LIN {X 0,Y 312.008,Z 393.675,A -85,B 0,C 180,E1 -15970.642,E2 -15970.642} C_VEL
LIN {X 0,Y 309.951,Z 389.912,A -85,B 0,C 180,E1 -15971.165,E2 -15971.165} C_VEL
LIN {X 0,Y 307.208,Z 381.469,A -85,B 0,C 180,E1 -15974.218,E2 -15974.218} C_VEL
LIN {X 0,Y 305.411,Z 376.065,A -85,B 0,C 180,E1 -15976.343,E2 -15976.343} C_VEL
LIN {X 0,Y 305.408,Z 376.064,A -85,B 0,C 180,E1 -15979.885,E2 -15979.885} C_VEL
LIN {X 0,Y 305.462,Z 376.035,A -85,B 0,C 180,E1 -15983.637,E2 -15983.637} C_VEL
LIN {X 0,Y 305.464,Z 376.059,A -85,B 0,C 180,E1 -15986.484,E2 -15986.484} C_VEL
LIN {X 0,Y 305.432,Z 376.032,A -85,B 0,C 180,E1 -15989.588,E2 -15989.588} C_VEL
LIN {X 0,Y 305.466,Z 376.057,A -85,B 0,C 180,E1 -15992.604,E2 -15992.604} C_VEL
LIN {X 0,Y 305.486,Z 376.057,A -85,B 0,C 180,E1 -15995.537,E2 -15995.537} C_VEL
LIN {X 0,Y 305.511,Z 376.05,A -85,B 0,C 180,E1 -15999.815,E2 -15999.815} C_VEL
LIN {X 0,Y 305.575,Z 376.046,A -85,B 0,C 180,E1 -16002.604,E2 -16002.604} C_VEL
LIN {X 0,Y 305.65,Z 376.036,A -85,B 0,C 180,E1 -16005.35,E2 -16005.35} C_VEL
LIN {X 0,Y 305.625,Z 376.039,A -85,B 0,C 180,E1 -16009.4,E2 -16009.4} C_VEL
LIN {X 0,Y 305.747,Z 376.015,A -85,B 0,C 180,E1 -16012.073,E2 -16012.073} C_VEL
LIN {X 0,Y 305.667,Z 376.028,A -85,B 0,C 180,E1 -16014.724,E2 -16014.724} C_VEL
LIN {X 0,Y 305.941,Z 375.994,A -85,B 0,C 180,E1 -16018.684,E2 -16018.684} C_VEL
LIN {X 0,Y 305.949,Z 376,A -85,B 0,C 180,E1 -16021.317,E2 -16021.317} C_VEL
LIN {X 0,Y 305.789,Z 376.012,A -85,B 0,C 180,E1 -16026.599,E2 -16026.599} C_VEL
LIN {X 0,Y 305.7,Z 376.031,A -85,B 0,C 180,E1 -16029.261,E2 -16029.261} C_VEL
LIN {X 0,Y 305.592,Z 376.043,A -85,B 0,C 180,E1 -16033.297,E2 -16033.297} C_VEL
LIN {X 0,Y 305.596,Z 376.042,A -85,B 0,C 180,E1 -16036.021,E2 -16036.021} C_VEL
LIN {X 0,Y 305.563,Z 376.014,A -85,B 0,C 180,E1 -16039.437,E2 -16039.437} C_VEL
LIN {X 0,Y 305.457,Z 376.061,A -85,B 0,C 180,E1 -16043.026,E2 -16043.026} C_VEL
LIN {X 0,Y 305.459,Z 376.033,A -85,B 0,C 180,E1 -16046.193,E2 -16046.193} C_VEL
LIN {X 0,Y 305.465,Z 376.058,A -85,B 0,C 180,E1 -16049.039,E2 -16049.039} C_VEL
LIN {X 0,Y 305.439,Z 376.045,A -85,B 0,C 180,E1 -16051.953,E2 -16051.953} C_VEL
LIN {X 0,Y 305.463,Z 376.042,A -85,B 0,C 180,E1 -16055.114,E2 -16055.114} C_VEL
LIN {X 0,Y 305.458,Z 376.146,A -85,B 0,C 180,E1 -16057.778,E2 -16057.778} C_VEL
LIN {X 0,Y 305.692,Z 377.224,A -85,B 0,C 180,E1 -16058.109,E2 -16058.109} C_VEL
LIN {X 0,Y 307.128,Z 379.845,A -85,B 0,C 180,E1 -16058.474,E2 -16058.474} C_VEL
LIN {X 0,Y 309.196,Z 382.473,A -85,B 0,C 180,E1 -16058.952,E2 -16058.952} C_VEL
LIN {X 0,Y 315.262,Z 391.574,A -85,B 0,C 180,E1 -16060.337,E2 -16060.337} C_VEL
LIN {X 0,Y 323.299,Z 404.841,A -85,B 0,C 180,E1 -16062.079,E2 -16062.079} C_VEL
LIN {X 0,Y 331.219,Z 419.433,A -85,B 0,C 180,E1 -16063.71,E2 -16063.71} C_VEL
LIN {X 0,Y 336.796,Z 430.906,A -85,B 0,C 180,E1 -16064.82,E2 -16064.82} C_VEL
LIN {X 0,Y 332.896,Z 525.367,A -85,B 0,C 180,E1 -16066.831,E2 -16066.831} C_VEL
LIN {X 0,Y 332.024,Z 544.302,A -85,B 0,C 180,E1 -16067.312,E2 -16067.312} C_VEL
LIN {X 0,Y 330.677,Z 559.768,A -85,B 0,C 180,E1 -16067.932,E2 -16067.932} C_VEL
LIN {X 0,Y 329.028,Z 573.938,A -85,B 0,C 180,E1 -16068.739,E2 -16068.739} C_VEL
LIN {X 0,Y 326.677,Z 588.476,A -85,B 0,C 180,E1 -16069.804,E2 -16069.804} C_VEL
LIN {X 0,Y 324.399,Z 601.799,A -85,B 0,C 180,E1 -16071.077,E2 -16071.077} C_VEL
LIN {X 0,Y 321.786,Z 614.094,A -85,B 0,C 180,E1 -16072.497,E2 -16072.497} C_VEL
LIN {X 0,Y 319.107,Z 625.525,A -85,B 0,C 180,E1 -16074.099,E2 -16074.099} C_VEL
LIN {X 0,Y 316.387,Z 636.114,A -85,B 0,C 180,E1 -16075.889,E2 -16075.889} C_VEL
LIN {X 0,Y 313.466,Z 647.104,A -85,B 0,C 180,E1 -16078.154,E2 -16078.154} C_VEL
LIN {X 0,Y 310.816,Z 656.515,A -85,B 0,C 180,E1 -16080.541,E2 -16080.541} C_VEL
LIN {X 0,Y 308.727,Z 664.118,A -85,B 0,C 180,E1 -16082.916,E2 -16082.916} C_VEL
LIN {X 0,Y 306.792,Z 671.137,A -85,B 0,C 180,E1 -16085.648,E2 -16085.648} C_VEL
LIN {X 0,Y 305.382,Z 676.578,A -85,B 0,C 180,E1 -16088.394,E2 -16088.394} C_VEL
LIN {X 0,Y 304.506,Z 680.595,A -85,B 0,C 180,E1 -16091.148,E2 -16091.148} C_VEL
LIN {X 0,Y 303.877,Z 683.314,A -85,B 0,C 180,E1 -16093.887,E2 -16093.887} C_VEL
LIN {X 0,Y 303.662,Z 684.816,A -85,B 0,C 180,E1 -16096.618,E2 -16096.618} C_VEL
LIN {X 0,Y 303.427,Z 685.154,A -85,B 0,C 180,E1 -16099.322,E2 -16099.322} C_VEL
LIN {X 0,Y 303.481,Z 684.345,A -85,B 0,C 180,E1 -16102.013,E2 -16102.013} C_VEL
LIN {X 0,Y 303.749,Z 682.375,A -85,B 0,C 180,E1 -16104.69,E2 -16104.69} C_VEL
LIN {X 0,Y 303.979,Z 679.192,A -85,B 0,C 180,E1 -16107.35,E2 -16107.35} C_VEL
LIN {X 0,Y 304.483,Z 674.772,A -85,B 0,C 180,E1 -16110,E2 -16110} C_VEL
LIN {X 0,Y 305.284,Z 669.021,A -85,B 0,C 180,E1 -16112.639,E2 -16112.639} C_VEL
LIN {X 0,Y 306.568,Z 661.77,A -85,B 0,C 180,E1 -16115.261,E2 -16115.261} C_VEL
LIN {X 0,Y 308.121,Z 654.006,A -85,B 0,C 180,E1 -16117.536,E2 -16117.536} C_VEL
LIN {X 0,Y 309.891,Z 644.712,A -85,B 0,C 180,E1 -16119.793,E2 -16119.793} C_VEL
LIN {X 0,Y 311.707,Z 635.269,A -85,B 0,C 180,E1 -16121.708,E2 -16121.708} C_VEL
LIN {X 0,Y 313.915,Z 624.043,A -85,B 0,C 180,E1 -16123.596,E2 -16123.596} C_VEL
LIN {X 0,Y 315.97,Z 611.759,A -85,B 0,C 180,E1 -16125.315,E2 -16125.315} C_VEL
LIN {X 0,Y 318.171,Z 598.17,A -85,B 0,C 180,E1 -16126.853,E2 -16126.853} C_VEL
LIN {X 0,Y 319.993,Z 584.854,A -85,B 0,C 180,E1 -16128.073,E2 -16128.073} C_VEL
LIN {X 0,Y 321.678,Z 570.085,A -85,B 0,C 180,E1 -16129.131,E2 -16129.131} C_VEL
LIN {X 0,Y 323.055,Z 555.393,A -85,B 0,C 180,E1 -16129.914,E2 -16129.914} C_VEL
LIN {X 0,Y 323.925,Z 540.407,A -85,B 0,C 180,E1 -16130.479,E2 -16130.479} C_VEL
LIN {X 0,Y 327.674,Z 425.087,A -85,B 0,C 180,E1 -16133.005,E2 -16133.005} C_VEL
LIN {X 0,Y 327.355,Z 423.116,A -85,B 0,C 180,E1 -16133.086,E2 -16133.086} C_VEL
LIN {X 0,Y 319.54,Z 404.611,A -85,B 0,C 180,E1 -16134.363,E2 -16134.363} C_VEL
LIN {X 0,Y 311.06,Z 386.835,A -85,B 0,C 180,E1 -16135.777,E2 -16135.777} C_VEL
LIN {X 0,Y 306.672,Z 379.243,A -85,B 0,C 180,E1 -16136.503,E2 -16136.503} C_VEL
LIN {X 0,Y 305.851,Z 377.64,A -85,B 0,C 180,E1 -16136.647,E2 -16136.647} C_VEL
LIN {X 0,Y 305.049,Z 376.531,A -85,B 0,C 180,E1 -16136.872,E2 -16136.872} C_VEL
LIN {X 0,Y 303.78,Z 376.27,A -85,B 0,C 180,E1 -16137.343,E2 -16137.343} C_VEL
LIN {X 0,Y 300.721,Z 376.645,A -85,B 0,C 180,E1 -16139.038,E2 -16139.038} C_VEL
LIN {X 0,Y 299.352,Z 377.162,A -85,B 0,C 180,E1 -16140.301,E2 -16140.301} C_VEL
LIN {X 0,Y 298.388,Z 376.931,A -85,B 0,C 180,E1 -16142.464,E2 -16142.464} C_VEL
LIN {X 0,Y 298.409,Z 376.927,A -85,B 0,C 180,E1 -16146.071,E2 -16146.071} C_VEL
LIN {X 0,Y 298.377,Z 376.934,A -85,B 0,C 180,E1 -16149.491,E2 -16149.491} C_VEL
LIN {X 0,Y 298.403,Z 376.94,A -85,B 0,C 180,E1 -16153.103,E2 -16153.103} C_VEL
LIN {X 0,Y 298.374,Z 376.928,A -85,B 0,C 180,E1 -16156.915,E2 -16156.915} C_VEL
LIN {X 0,Y 298.354,Z 376.938,A -85,B 0,C 180,E1 -16161.019,E2 -16161.019} C_VEL
LIN {X 0,Y 298.407,Z 376.939,A -85,B 0,C 180,E1 -16163.928,E2 -16163.928} C_VEL
LIN {X 0,Y 298.396,Z 376.937,A -85,B 0,C 180,E1 -16167.199,E2 -16167.199} C_VEL
LIN {X 0,Y 298.404,Z 376.927,A -85,B 0,C 180,E1 -16170.625,E2 -16170.625} C_VEL
LIN {X 0,Y 298.416,Z 376.89,A -85,B 0,C 180,E1 -16174.917,E2 -16174.917} C_VEL
LIN {X 0,Y 298.429,Z 376.937,A -85,B 0,C 180,E1 -16179.313,E2 -16179.313} C_VEL
LIN {X 0,Y 298.508,Z 376.909,A -85,B 0,C 180,E1 -16182.177,E2 -16182.177} C_VEL
LIN {X 0,Y 298.588,Z 376.913,A -85,B 0,C 180,E1 -16184.994,E2 -16184.994} C_VEL
LIN {X 0,Y 298.586,Z 376.897,A -85,B 0,C 180,E1 -16189.146,E2 -16189.146} C_VEL
LIN {X 0,Y 298.7,Z 376.901,A -85,B 0,C 180,E1 -16191.884,E2 -16191.884} C_VEL
LIN {X 0,Y 298.63,Z 376.893,A -85,B 0,C 180,E1 -16194.598,E2 -16194.598} C_VEL
LIN {X 0,Y 298.915,Z 376.873,A -85,B 0,C 180,E1 -16198.652,E2 -16198.652} C_VEL
LIN {X 0,Y 298.909,Z 376.859,A -85,B 0,C 180,E1 -16201.347,E2 -16201.347} C_VEL
LIN {X 0,Y 298.635,Z 376.912,A -85,B 0,C 180,E1 -16205.401,E2 -16205.401} C_VEL
LIN {X 0,Y 298.709,Z 376.893,A -85,B 0,C 180,E1 -16208.819,E2 -16208.819} C_VEL
LIN {X 0,Y 298.545,Z 376.911,A -85,B 0,C 180,E1 -16212.231,E2 -16212.231} C_VEL
LIN {X 0,Y 298.524,Z 376.92,A -85,B 0,C 180,E1 -16215.15,E2 -16215.15} C_VEL
LIN {X 0,Y 298.499,Z 376.923,A -85,B 0,C 180,E1 -16219.647,E2 -16219.647} C_VEL
LIN {X 0,Y 298.424,Z 376.932,A -85,B 0,C 180,E1 -16223.6,E2 -16223.6} C_VEL
LIN {X 0,Y 298.408,Z 376.931,A -85,B 0,C 180,E1 -16226.582,E2 -16226.582} C_VEL
LIN {X 0,Y 298.394,Z 376.936,A -85,B 0,C 180,E1 -16229.643,E2 -16229.643} C_VEL
LIN {X 0,Y 298.392,Z 376.937,A -85,B 0,C 180,E1 -16232.8,E2 -16232.8} C_VEL
LIN {X 0,Y 298.426,Z 376.935,A -85,B 0,C 180,E1 -16236.802,E2 -16236.802} C_VEL
LIN {X 0,Y 298.347,Z 376.945,A -85,B 0,C 180,E1 -16241.267,E2 -16241.267} C_VEL
LIN {X 0,Y 298.353,Z 376.946,A -85,B 0,C 180,E1 -16245.034,E2 -16245.034} C_VEL
LIN {X 0,Y 298.378,Z 377.05,A -85,B 0,C 180,E1 -16248.765,E2 -16248.765} C_VEL
LIN {X 0,Y 301.352,Z 387.503,A -85,B 0,C 180,E1 -16251.914,E2 -16251.914} C_VEL
LIN {X 0,Y 302.25,Z 391.009,A -85,B 0,C 180,E1 -16252.878,E2 -16252.878} C_VEL
LIN {X 0,Y 310.107,Z 407.933,A -85,B 0,C 180,E1 -16254.276,E2 -16254.276} C_VEL
LIN {X 0,Y 317.769,Z 426.003,A -85,B 0,C 180,E1 -16255.596,E2 -16255.596} C_VEL
LIN {X 0,Y 318.599,Z 429.317,A -85,B 0,C 180,E1 -16255.77,E2 -16255.77} C_VEL
LIN {X 0,Y 321.034,Z 444.923,A -85,B 0,C 180,E1 -16256.421,E2 -16256.421} C_VEL
LIN {X 0,Y 317.296,Z 558.27,A -85,B 0,C 180,E1 -16258.957,E2 -16258.957} C_VEL
LIN {X 0,Y 316.142,Z 573.476,A -85,B 0,C 180,E1 -16259.527,E2 -16259.527} C_VEL
LIN {X 0,Y 314.609,Z 587.681,A -85,B 0,C 180,E1 -16260.288,E2 -16260.288} C_VEL
LIN {X 0,Y 312.776,Z 601.94,A -85,B 0,C 180,E1 -16261.309,E2 -16261.309} C_VEL
LIN {X 0,Y 310.741,Z 615.574,A -85,B 0,C 180,E1 -16262.56,E2 -16262.56} C_VEL
LIN {X 0,Y 308.581,Z 628.233,A -85,B 0,C 180,E1 -16263.997,E2 -16263.997} C_VEL
LIN {X 0,Y 306.139,Z 641.062,A -85,B 0,C 180,E1 -16265.773,E2 -16265.773} C_VEL
LIN {X 0,Y 304.1,Z 651.792,A -85,B 0,C 180,E1 -16267.582,E2 -16267.582} C_VEL
LIN {X 0,Y 302.25,Z 661.737,A -85,B 0,C 180,E1 -16269.587,E2 -16269.587} C_VEL
LIN {X 0,Y 300.332,Z 671.446,A -85,B 0,C 180,E1 -16271.937,E2 -16271.937} C_VEL
LIN {X 0,Y 298.89,Z 679.527,A -85,B 0,C 180,E1 -16274.312,E2 -16274.312} C_VEL
LIN {X 0,Y 297.746,Z 687.046,A -85,B 0,C 180,E1 -16277.042,E2 -16277.042} C_VEL
LIN {X 0,Y 296.974,Z 692.994,A -85,B 0,C 180,E1 -16279.776,E2 -16279.776} C_VEL
LIN {X 0,Y 296.719,Z 696.522,A -85,B 0,C 180,E1 -16281.83,E2 -16281.83} C_VEL
LIN {X 0,Y 296.549,Z 700.073,A -85,B 0,C 180,E1 -16284.56,E2 -16284.56} C_VEL
LIN {X 0,Y 296.54,Z 702.389,A -85,B 0,C 180,E1 -16287.283,E2 -16287.283} C_VEL
LIN {X 0,Y 296.533,Z 703.529,A -85,B 0,C 180,E1 -16290,E2 -16290} C_VEL
LIN {X 0,Y 296.525,Z 703.493,A -85,B 0,C 180,E1 -16292.717,E2 -16292.717} C_VEL
LIN {X 0,Y 296.51,Z 702.276,A -85,B 0,C 180,E1 -16295.44,E2 -16295.44} C_VEL
LIN {X 0,Y 296.704,Z 699.922,A -85,B 0,C 180,E1 -16298.171,E2 -16298.171} C_VEL
LIN {X 0,Y 297.218,Z 696.389,A -85,B 0,C 180,E1 -16300.904,E2 -16300.904} C_VEL
LIN {X 0,Y 298.236,Z 691.598,A -85,B 0,C 180,E1 -16303.63,E2 -16303.63} C_VEL
LIN {X 0,Y 299.688,Z 685.423,A -85,B 0,C 180,E1 -16306.345,E2 -16306.345} C_VEL
LIN {X 0,Y 301.786,Z 677.699,A -85,B 0,C 180,E1 -16309.028,E2 -16309.028} C_VEL
LIN {X 0,Y 304.1,Z 669.495,A -85,B 0,C 180,E1 -16311.346,E2 -16311.346} C_VEL
LIN {X 0,Y 306.627,Z 660.122,A -85,B 0,C 180,E1 -16313.536,E2 -16313.536} C_VEL
LIN {X 0,Y 309.527,Z 649.618,A -85,B 0,C 180,E1 -16315.557,E2 -16315.557} C_VEL
LIN {X 0,Y 312.649,Z 637.725,A -85,B 0,C 180,E1 -16317.44,E2 -16317.44} C_VEL
LIN {X 0,Y 315.537,Z 625.876,A -85,B 0,C 180,E1 -16318.976,E2 -16318.976} C_VEL
LIN {X 0,Y 318.347,Z 613.086,A -85,B 0,C 180,E1 -16320.331,E2 -16320.331} C_VEL
LIN {X 0,Y 320.902,Z 599.132,A -85,B 0,C 180,E1 -16321.527,E2 -16321.527} C_VEL
LIN {X 0,Y 323.175,Z 584.768,A -85,B 0,C 180,E1 -16322.471,E2 -16322.471} C_VEL
LIN {X 0,Y 325.045,Z 570.002,A -85,B 0,C 180,E1 -16323.182,E2 -16323.182} C_VEL
LIN {X 0,Y 326.354,Z 554.891,A -85,B 0,C 180,E1 -16323.678,E2 -16323.678} C_VEL
LIN {X 0,Y 330.69,Z 446.764,A -85,B 0,C 180,E1 -16326.074,E2 -16326.074} C_VEL
LIN {X 0,Y 329.355,Z 439.216,A -85,B 0,C 180,E1 -16326.478,E2 -16326.478} C_VEL
LIN {X 0,Y 321.063,Z 421.84,A -85,B 0,C 180,E1 -16328.245,E2 -16328.245} C_VEL
LIN {X 0,Y 312.778,Z 406.54,A -85,B 0,C 180,E1 -16330.1,E2 -16330.1} C_VEL
LIN {X 0,Y 307.454,Z 397.794,A -85,B 0,C 180,E1 -16331.344,E2 -16331.344} C_VEL
LIN {X 0,Y 305.141,Z 394.014,A -85,B 0,C 180,E1 -16331.907,E2 -16331.907} C_VEL
LIN {X 0,Y 302.575,Z 389.595,A -85,B 0,C 180,E1 -16332.584,E2 -16332.584} C_VEL
LIN {X 0,Y 299.446,Z 380.298,A -85,B 0,C 180,E1 -16336.184,E2 -16336.184} C_VEL
LIN {X 0,Y 298.4,Z 376.939,A -85,B 0,C 180,E1 -16337.61,E2 -16337.61} C_VEL
LIN {X 0,Y 298.384,Z 376.941,A -85,B 0,C 180,E1 -16341.011,E2 -16341.011} C_VEL
LIN {X 0,Y 298.404,Z 376.913,A -85,B 0,C 180,E1 -16343.929,E2 -16343.929} C_VEL
LIN {X 0,Y 298.392,Z 376.931,A -85,B 0,C 180,E1 -16347.2,E2 -16347.2} C_VEL
LIN {X 0,Y 298.407,Z 376.917,A -85,B 0,C 180,E1 -16350.624,E2 -16350.624} C_VEL
LIN {X 0,Y 298.446,Z 376.934,A -85,B 0,C 180,E1 -16354.921,E2 -16354.921} C_VEL
LIN {X 0,Y 298.444,Z 376.933,A -85,B 0,C 180,E1 -16359.315,E2 -16359.315} C_VEL
LIN {X 0,Y 298.535,Z 376.924,A -85,B 0,C 180,E1 -16362.18,E2 -16362.18} C_VEL
LIN {X 0,Y 298.594,Z 376.911,A -85,B 0,C 180,E1 -16364.995,E2 -16364.995} C_VEL
LIN {X 0,Y 298.584,Z 376.917,A -85,B 0,C 180,E1 -16369.147,E2 -16369.147} C_VEL
LIN {X 0,Y 298.699,Z 376.892,A -85,B 0,C 180,E1 -16371.885,E2 -16371.885} C_VEL
LIN {X 0,Y 298.636,Z 376.905,A -85,B 0,C 180,E1 -16374.599,E2 -16374.599} C_VEL
LIN {X 0,Y 298.91,Z 376.87,A -85,B 0,C 180,E1 -16378.653,E2 -16378.653} C_VEL
LIN {X 0,Y 298.916,Z 376.876,A -85,B 0,C 180,E1 -16381.348,E2 -16381.348} C_VEL
LIN {X 0,Y 298.737,Z 376.889,A -85,B 0,C 180,E1 -16386.756,E2 -16386.756} C_VEL
LIN {X 0,Y 298.632,Z 376.911,A -85,B 0,C 180,E1 -16389.483,E2 -16389.483} C_VEL
LIN {X 0,Y 298.555,Z 376.92,A -85,B 0,C 180,E1 -16393.616,E2 -16393.616} C_VEL
LIN {X 0,Y 298.551,Z 376.923,A -85,B 0,C 180,E1 -16396.409,E2 -16396.409} C_VEL
LIN {X 0,Y 298.496,Z 376.893,A -85,B 0,C 180,E1 -16399.646,E2 -16399.646} C_VEL
LIN {X 0,Y 298.386,Z 376.936,A -85,B 0,C 180,E1 -16403.604,E2 -16403.604} C_VEL
LIN {X 0,Y 298.407,Z 376.913,A -85,B 0,C 180,E1 -16406.583,E2 -16406.583} C_VEL
LIN {X 0,Y 298.402,Z 376.926,A -85,B 0,C 180,E1 -16409.644,E2 -16409.644} C_VEL
LIN {X 0,Y 298.395,Z 376.935,A -85,B 0,C 180,E1 -16412.801,E2 -16412.801} C_VEL
LIN {X 0,Y 298.418,Z 376.96,A -85,B 0,C 180,E1 -16416.53,E2 -16416.53} C_VEL
LIN {X 0,Y 298.525,Z 377.581,A -85,B 0,C 180,E1 -16416.669,E2 -16416.669} C_VEL
LIN {X 0,Y 299.706,Z 380.222,A -85,B 0,C 180,E1 -16417.009,E2 -16417.009} C_VEL
LIN {X 0,Y 301.827,Z 382.507,A -85,B 0,C 180,E1 -16417.521,E2 -16417.521} C_VEL
LIN {X 0,Y 303.801,Z 385.631,A -85,B 0,C 180,E1 -16418.021,E2 -16418.021} C_VEL
LIN {X 0,Y 305.3,Z 387.534,A -85,B 0,C 180,E1 -16418.377,E2 -16418.377} C_VEL
LIN {X 0,Y 311.863,Z 397.674,A -85,B 0,C 180,E1 -16419.928,E2 -16419.928} C_VEL
LIN {X 0,Y 319.09,Z 409.756,A -85,B 0,C 180,E1 -16421.543,E2 -16421.543} C_VEL
LIN {X 0,Y 326.096,Z 422.733,A -85,B 0,C 180,E1 -16423.036,E2 -16423.036} C_VEL
LIN {X 0,Y 331.26,Z 433.44,A -85,B 0,C 180,E1 -16424.107,E2 -16424.107} C_VEL
LIN {X 0,Y 327.037,Z 530.162,A -85,B 0,C 180,E1 -16426.181,E2 -16426.181} C_VEL
LIN {X 0,Y 326.245,Z 546.715,A -85,B 0,C 180,E1 -16426.652,E2 -16426.652} C_VEL
LIN {X 0,Y 324.83,Z 561.215,A -85,B 0,C 180,E1 -16427.262,E2 -16427.262} C_VEL
LIN {X 0,Y 323.026,Z 575.6,A -85,B 0,C 180,E1 -16428.113,E2 -16428.113} C_VEL
LIN {X 0,Y 320.758,Z 588.911,A -85,B 0,C 180,E1 -16429.112,E2 -16429.112} C_VEL
LIN {X 0,Y 318.366,Z 602.299,A -85,B 0,C 180,E1 -16430.416,E2 -16430.416} C_VEL
LIN {X 0,Y 315.67,Z 614.443,A -85,B 0,C 180,E1 -16431.843,E2 -16431.843} C_VEL
LIN {X 0,Y 312.879,Z 625.846,A -85,B 0,C 180,E1 -16433.469,E2 -16433.469} C_VEL
LIN {X 0,Y 309.822,Z 637.27,A -85,B 0,C 180,E1 -16435.452,E2 -16435.452} C_VEL
LIN {X 0,Y 307.14,Z 646.858,A -85,B 0,C 180,E1 -16437.472,E2 -16437.472} C_VEL
LIN {X 0,Y 304.374,Z 656.187,A -85,B 0,C 180,E1 -16439.854,E2 -16439.854} C_VEL
LIN {X 0,Y 302.142,Z 663.872,A -85,B 0,C 180,E1 -16442.276,E2 -16442.276} C_VEL
LIN {X 0,Y 300.05,Z 670.989,A -85,B 0,C 180,E1 -16445.064,E2 -16445.064} C_VEL
LIN {X 0,Y 298.521,Z 676.514,A -85,B 0,C 180,E1 -16447.872,E2 -16447.872} C_VEL
LIN {X 0,Y 297.484,Z 680.892,A -85,B 0,C 180,E1 -16450.91,E2 -16450.91} C_VEL
LIN {X 0,Y 296.846,Z 683.406,A -85,B 0,C 180,E1 -16453.495,E2 -16453.495} C_VEL
LIN {X 0,Y 296.569,Z 684.991,A -85,B 0,C 180,E1 -16456.317,E2 -16456.317} C_VEL
LIN {X 0,Y 296.356,Z 685.393,A -85,B 0,C 180,E1 -16459.064,E2 -16459.064} C_VEL
LIN {X 0,Y 296.39,Z 684.656,A -85,B 0,C 180,E1 -16461.821,E2 -16461.821} C_VEL
LIN {X 0,Y 296.648,Z 682.726,A -85,B 0,C 180,E1 -16464.562,E2 -16464.562} C_VEL
LIN {X 0,Y 296.882,Z 679.615,A -85,B 0,C 180,E1 -16467.286,E2 -16467.286} C_VEL
LIN {X 0,Y 297.402,Z 675.273,A -85,B 0,C 180,E1 -16470,E2 -16470} C_VEL
LIN {X 0,Y 298.221,Z 669.604,A -85,B 0,C 180,E1 -16472.702,E2 -16472.702} C_VEL
LIN {X 0,Y 299.523,Z 662.443,A -85,B 0,C 180,E1 -16475.386,E2 -16475.386} C_VEL
LIN {X 0,Y 301.111,Z 654.778,A -85,B 0,C 180,E1 -16477.713,E2 -16477.713} C_VEL
LIN {X 0,Y 302.956,Z 645.59,A -85,B 0,C 180,E1 -16480.02,E2 -16480.02} C_VEL
LIN {X 0,Y 304.813,Z 636.277,A -85,B 0,C 180,E1 -16481.977,E2 -16481.977} C_VEL
LIN {X 0,Y 307.091,Z 625.19,A -85,B 0,C 180,E1 -16483.904,E2 -16483.904} C_VEL
LIN {X 0,Y 309.222,Z 613.076,A -85,B 0,C 180,E1 -16485.658,E2 -16485.658} C_VEL
LIN {X 0,Y 311.462,Z 599.754,A -85,B 0,C 180,E1 -16487.227,E2 -16487.227} C_VEL
LIN {X 0,Y 313.592,Z 584.865,A -85,B 0,C 180,E1 -16488.624,E2 -16488.624} C_VEL
LIN {X 0,Y 315.309,Z 570.043,A -85,B 0,C 180,E1 -16489.702,E2 -16489.702} C_VEL
LIN {X 0,Y 316.741,Z 555.244,A -85,B 0,C 180,E1 -16490.497,E2 -16490.497} C_VEL
LIN {X 0,Y 317.652,Z 540.071,A -85,B 0,C 180,E1 -16491.071,E2 -16491.071} C_VEL
LIN {X 0,Y 321.482,Z 426.854,A -85,B 0,C 180,E1 -16493.589,E2 -16493.589} C_VEL
LIN {X 0,Y 321.068,Z 424.843,A -85,B 0,C 180,E1 -16493.683,E2 -16493.683} C_VEL
LIN {X 0,Y 313.395,Z 406.641,A -85,B 0,C 180,E1 -16494.983,E2 -16494.983} C_VEL
LIN {X 0,Y 305.579,Z 390.346,A -85,B 0,C 180,E1 -16496.33,E2 -16496.33} C_VEL
LIN {X 0,Y 299.769,Z 380.27,A -85,B 0,C 180,E1 -16497.331,E2 -16497.331} C_VEL
LIN {X 0,Y 298.5,Z 377.502,A -85,B 0,C 180,E1 -16497.573,E2 -16497.573} C_VEL
LIN {X 0,Y 298.421,Z 376.937,A -85,B 0,C 180,E1 -16497.619,E2 -16497.619} C_VEL
LIN {X 0,Y 298.382,Z 376.943,A -85,B 0,C 180,E1 -16501.211,E2 -16501.211} C_VEL
LIN {X 0,Y 298.388,Z 376.931,A -85,B 0,C 180,E1 -16502.464,E2 -16502.464} C_VEL
LIN {X 0,Y 297.729,Z 377.021,A -85,B 0,C 180,E1 -16503.59,E2 -16503.59} C_VEL
LIN {X 0,Y 294.858,Z 377.374,A -85,B 0,C 180,E1 -16505.422,E2 -16505.422} C_VEL
LIN {X 0,Y 292.426,Z 377.674,A -85,B 0,C 180,E1 -16506.909,E2 -16506.909} C_VEL
LIN {X 0,Y 291.398,Z 377.813,A -85,B 0,C 180,E1 -16508.062,E2 -16508.062} C_VEL
LIN {X 0,Y 291.323,Z 377.817,A -85,B 0,C 180,E1 -16508.452,E2 -16508.452} C_VEL
LIN {X 0,Y 291.291,Z 377.824,A -85,B 0,C 180,E1 -16512.498,E2 -16512.498} C_VEL
LIN {X 0,Y 291.292,Z 377.805,A -85,B 0,C 180,E1 -16516.37,E2 -16516.37} C_VEL
LIN {X 0,Y 291.313,Z 377.817,A -85,B 0,C 180,E1 -16520.535,E2 -16520.535} C_VEL
LIN {X 0,Y 291.388,Z 377.812,A -85,B 0,C 180,E1 -16522.916,E2 -16522.916} C_VEL
LIN {X 0,Y 291.346,Z 377.811,A -85,B 0,C 180,E1 -16526.301,E2 -16526.301} C_VEL
LIN {X 0,Y 291.367,Z 377.808,A -85,B 0,C 180,E1 -16530.268,E2 -16530.268} C_VEL
LIN {X 0,Y 291.344,Z 377.764,A -85,B 0,C 180,E1 -16534.264,E2 -16534.264} C_VEL
LIN {X 0,Y 291.354,Z 377.805,A -85,B 0,C 180,E1 -16537.297,E2 -16537.297} C_VEL
LIN {X 0,Y 291.442,Z 377.804,A -85,B 0,C 180,E1 -16540.268,E2 -16540.268} C_VEL
LIN {X 0,Y 291.517,Z 377.793,A -85,B 0,C 180,E1 -16544.652,E2 -16544.652} C_VEL
LIN {X 0,Y 291.532,Z 377.775,A -85,B 0,C 180,E1 -16548.88,E2 -16548.88} C_VEL
LIN {X 0,Y 291.654,Z 377.78,A -85,B 0,C 180,E1 -16551.686,E2 -16551.686} C_VEL
LIN {X 0,Y 291.6,Z 377.769,A -85,B 0,C 180,E1 -16554.467,E2 -16554.467} C_VEL
LIN {X 0,Y 291.881,Z 377.749,A -85,B 0,C 180,E1 -16558.62,E2 -16558.62} C_VEL
LIN {X 0,Y 291.877,Z 377.735,A -85,B 0,C 180,E1 -16561.379,E2 -16561.379} C_VEL
LIN {X 0,Y 291.605,Z 377.786,A -85,B 0,C 180,E1 -16565.532,E2 -16565.532} C_VEL
LIN {X 0,Y 291.668,Z 377.77,A -85,B 0,C 180,E1 -16568.909,E2 -16568.909} C_VEL
LIN {X 0,Y 291.509,Z 377.786,A -85,B 0,C 180,E1 -16572.531,E2 -16572.531} C_VEL
LIN {X 0,Y 291.461,Z 377.801,A -85,B 0,C 180,E1 -16575.381,E2 -16575.381} C_VEL
LIN {X 0,Y 291.452,Z 377.804,A -85,B 0,C 180,E1 -16579.874,E2 -16579.874} C_VEL
LIN {X 0,Y 291.364,Z 377.814,A -85,B 0,C 180,E1 -16584.208,E2 -16584.208} C_VEL
LIN {X 0,Y 291.354,Z 377.813,A -85,B 0,C 180,E1 -16587.278,E2 -16587.278} C_VEL
LIN {X 0,Y 291.319,Z 377.819,A -85,B 0,C 180,E1 -16590.438,E2 -16590.438} C_VEL
LIN {X 0,Y 291.343,Z 377.817,A -85,B 0,C 180,E1 -16593.698,E2 -16593.698} C_VEL
LIN {X 0,Y 291.353,Z 377.819,A -85,B 0,C 180,E1 -16597.247,E2 -16597.247} C_VEL
LIN {X 0,Y 291.294,Z 377.827,A -85,B 0,C 180,E1 -16601.588,E2 -16601.588} C_VEL
LIN {X 0,Y 291.281,Z 377.828,A -85,B 0,C 180,E1 -16605.596,E2 -16605.596} C_VEL
LIN {X 0,Y 291.296,Z 377.972,A -85,B 0,C 180,E1 -16608.025,E2 -16608.025} C_VEL
LIN {X 0,Y 294.876,Z 390.443,A -85,B 0,C 180,E1 -16611.898,E2 -16611.898} C_VEL
LIN {X 0,Y 302.989,Z 407.643,A -85,B 0,C 180,E1 -16613.431,E2 -16613.431} C_VEL
LIN {X 0,Y 311.672,Z 428.036,A -85,B 0,C 180,E1 -16614.988,E2 -16614.988} C_VEL
LIN {X 0,Y 312.61,Z 431.286,A -85,B 0,C 180,E1 -16615.178,E2 -16615.178} C_VEL
LIN {X 0,Y 314.848,Z 446.336,A -85,B 0,C 180,E1 -16615.813,E2 -16615.813} C_VEL
LIN {X 0,Y 311.077,Z 556.664,A -85,B 0,C 180,E1 -16618.313,E2 -16618.313} C_VEL
LIN {X 0,Y 309.886,Z 572.373,A -85,B 0,C 180,E1 -16618.891,E2 -16618.891} C_VEL
LIN {X 0,Y 308.238,Z 587.447,A -85,B 0,C 180,E1 -16619.704,E2 -16619.704} C_VEL
LIN {X 0,Y 306.264,Z 602.414,A -85,B 0,C 180,E1 -16620.801,E2 -16620.801} C_VEL
LIN {X 0,Y 304.12,Z 616.148,A -85,B 0,C 180,E1 -16622.098,E2 -16622.098} C_VEL
LIN {X 0,Y 301.895,Z 628.662,A -85,B 0,C 180,E1 -16623.562,E2 -16623.562} C_VEL
LIN {X 0,Y 299.377,Z 641.38,A -85,B 0,C 180,E1 -16625.374,E2 -16625.374} C_VEL
LIN {X 0,Y 297.067,Z 653.282,A -85,B 0,C 180,E1 -16627.46,E2 -16627.46} C_VEL
LIN {X 0,Y 294.895,Z 664.155,A -85,B 0,C 180,E1 -16629.783,E2 -16629.783} C_VEL
LIN {X 0,Y 293.024,Z 673.417,A -85,B 0,C 180,E1 -16632.194,E2 -16632.194} C_VEL
LIN {X 0,Y 291.593,Z 681.097,A -85,B 0,C 180,E1 -16634.626,E2 -16634.626} C_VEL
LIN {X 0,Y 290.51,Z 688.262,A -85,B 0,C 180,E1 -16637.424,E2 -16637.424} C_VEL
LIN {X 0,Y 289.812,Z 693.883,A -85,B 0,C 180,E1 -16640.227,E2 -16640.227} C_VEL
LIN {X 0,Y 289.548,Z 698.128,A -85,B 0,C 180,E1 -16643.029,E2 -16643.029} C_VEL
LIN {X 0,Y 289.415,Z 701.092,A -85,B 0,C 180,E1 -16645.822,E2 -16645.822} C_VEL
LIN {X 0,Y 289.431,Z 702.855,A -85,B 0,C 180,E1 -16648.609,E2 -16648.609} C_VEL
LIN {X 0,Y 289.424,Z 703.445,A -85,B 0,C 180,E1 -16651.391,E2 -16651.391} C_VEL
LIN {X 0,Y 289.378,Z 702.835,A -85,B 0,C 180,E1 -16654.178,E2 -16654.178} C_VEL
LIN {X 0,Y 289.465,Z 701.092,A -85,B 0,C 180,E1 -16656.973,E2 -16656.973} C_VEL
LIN {X 0,Y 289.894,Z 698.198,A -85,B 0,C 180,E1 -16659.771,E2 -16659.771} C_VEL
LIN {X 0,Y 290.719,Z 694.093,A -85,B 0,C 180,E1 -16662.566,E2 -16662.566} C_VEL
LIN {X 0,Y 291.955,Z 688.673,A -85,B 0,C 180,E1 -16665.355,E2 -16665.355} C_VEL
LIN {X 0,Y 293.86,Z 681.794,A -85,B 0,C 180,E1 -16668.114,E2 -16668.114} C_VEL
LIN {X 0,Y 296.288,Z 673.27,A -85,B 0,C 180,E1 -16670.843,E2 -16670.843} C_VEL
LIN {X 0,Y 299.079,Z 664.241,A -85,B 0,C 180,E1 -16673.179,E2 -16673.179} C_VEL
LIN {X 0,Y 302.116,Z 653.401,A -85,B 0,C 180,E1 -16675.49,E2 -16675.49} C_VEL
LIN {X 0,Y 305.53,Z 641.247,A -85,B 0,C 180,E1 -16677.576,E2 -16677.576} C_VEL
LIN {X 0,Y 308.804,Z 628.888,A -85,B 0,C 180,E1 -16679.295,E2 -16679.295} C_VEL
LIN {X 0,Y 311.95,Z 615.255,A -85,B 0,C 180,E1 -16680.833,E2 -16680.833} C_VEL
LIN {X 0,Y 314.586,Z 601.949,A -85,B 0,C 180,E1 -16682.042,E2 -16682.042} C_VEL
LIN {X 0,Y 317.062,Z 587.18,A -85,B 0,C 180,E1 -16683.082,E2 -16683.082} C_VEL
LIN {X 0,Y 319.228,Z 571.663,A -85,B 0,C 180,E1 -16683.867,E2 -16683.867} C_VEL
LIN {X 0,Y 320.534,Z 557.59,A -85,B 0,C 180,E1 -16684.374,E2 -16684.374} C_VEL
LIN {X 0,Y 324.931,Z 456.72,A -85,B 0,C 180,E1 -16686.636,E2 -16686.636} C_VEL
LIN {X 0,Y 325.143,Z 447.815,A -85,B 0,C 180,E1 -16686.858,E2 -16686.858} C_VEL
LIN {X 0,Y 324.162,Z 442.286,A -85,B 0,C 180,E1 -16687.165,E2 -16687.165} C_VEL
LIN {X 0,Y 316.397,Z 425.856,A -85,B 0,C 180,E1 -16688.886,E2 -16688.886} C_VEL
LIN {X 0,Y 307.885,Z 410.002,A -85,B 0,C 180,E1 -16690.868,E2 -16690.868} C_VEL
LIN {X 0,Y 301.204,Z 398.985,A -85,B 0,C 180,E1 -16692.511,E2 -16692.511} C_VEL
LIN {X 0,Y 297.725,Z 393.523,A -85,B 0,C 180,E1 -16693.407,E2 -16693.407} C_VEL
LIN {X 0,Y 295.168,Z 389.285,A -85,B 0,C 180,E1 -16694.12,E2 -16694.12} C_VEL
LIN {X 0,Y 292.297,Z 380.589,A -85,B 0,C 180,E1 -16697.684,E2 -16697.684} C_VEL
LIN {X 0,Y 291.313,Z 377.823,A -85,B 0,C 180,E1 -16698.955,E2 -16698.955} C_VEL
LIN {X 0,Y 291.389,Z 377.791,A -85,B 0,C 180,E1 -16702.917,E2 -16702.917} C_VEL
LIN {X 0,Y 291.343,Z 377.818,A -85,B 0,C 180,E1 -16706.302,E2 -16706.302} C_VEL
LIN {X 0,Y 291.368,Z 377.788,A -85,B 0,C 180,E1 -16710.267,E2 -16710.267} C_VEL
LIN {X 0,Y 291.373,Z 377.808,A -85,B 0,C 180,E1 -16714.268,E2 -16714.268} C_VEL
LIN {X 0,Y 291.377,Z 377.807,A -85,B 0,C 180,E1 -16717.3,E2 -16717.3} C_VEL
LIN {X 0,Y 291.458,Z 377.797,A -85,B 0,C 180,E1 -16720.271,E2 -16720.271} C_VEL
LIN {X 0,Y 291.556,Z 377.785,A -85,B 0,C 180,E1 -16724.624,E2 -16724.624} C_VEL
LIN {X 0,Y 291.53,Z 377.791,A -85,B 0,C 180,E1 -16728.881,E2 -16728.881} C_VEL
LIN {X 0,Y 291.652,Z 377.77,A -85,B 0,C 180,E1 -16731.687,E2 -16731.687} C_VEL
LIN {X 0,Y 291.605,Z 377.782,A -85,B 0,C 180,E1 -16734.468,E2 -16734.468} C_VEL
LIN {X 0,Y 291.877,Z 377.746,A -85,B 0,C 180,E1 -16738.621,E2 -16738.621} C_VEL
LIN {X 0,Y 291.882,Z 377.752,A -85,B 0,C 180,E1 -16741.38,E2 -16741.38} C_VEL
LIN {X 0,Y 291.689,Z 377.766,A -85,B 0,C 180,E1 -16746.92,E2 -16746.92} C_VEL
LIN {X 0,Y 291.574,Z 377.791,A -85,B 0,C 180,E1 -16749.714,E2 -16749.714} C_VEL
LIN {X 0,Y 291.525,Z 377.791,A -85,B 0,C 180,E1 -16753.951,E2 -16753.951} C_VEL
LIN {X 0,Y 291.489,Z 377.8,A -85,B 0,C 180,E1 -16756.818,E2 -16756.818} C_VEL
LIN {X 0,Y 291.453,Z 377.769,A -85,B 0,C 180,E1 -16759.875,E2 -16759.875} C_VEL
LIN {X 0,Y 291.331,Z 377.803,A -85,B 0,C 180,E1 -16764.212,E2 -16764.212} C_VEL
LIN {X 0,Y 291.358,Z 377.8,A -85,B 0,C 180,E1 -16767.279,E2 -16767.279} C_VEL
LIN {X 0,Y 291.324,Z 377.799,A -85,B 0,C 180,E1 -16770.439,E2 -16770.439} C_VEL
LIN {X 0,Y 291.346,Z 377.817,A -85,B 0,C 180,E1 -16773.699,E2 -16773.699} C_VEL
LIN {X 0,Y 291.367,Z 377.798,A -85,B 0,C 180,E1 -16775.09,E2 -16775.09} C_VEL
LIN {X 0,Y 292.259,Z 380.448,A -85,B 0,C 180,E1 -16775.408,E2 -16775.408} C_VEL
LIN {X 0,Y 294.223,Z 382.651,A -85,B 0,C 180,E1 -16775.925,E2 -16775.925} C_VEL
LIN {X 0,Y 295.005,Z 383.633,A -85,B 0,C 180,E1 -16776.131,E2 -16776.131} C_VEL
LIN {X 0,Y 297.166,Z 386.864,A -85,B 0,C 180,E1 -16776.71,E2 -16776.71} C_VEL
LIN {X 0,Y 298.394,Z 388.421,A -85,B 0,C 180,E1 -16777.022,E2 -16777.022} C_VEL
LIN {X 0,Y 304.326,Z 396.873,A -85,B 0,C 180,E1 -16778.499,E2 -16778.499} C_VEL
LIN {X 0,Y 313.192,Z 411.603,A -85,B 0,C 180,E1 -16780.6,E2 -16780.6} C_VEL
LIN {X 0,Y 320.534,Z 425.111,A -85,B 0,C 180,E1 -16782.236,E2 -16782.236} C_VEL
LIN {X 0,Y 325.707,Z 435.732,A -85,B 0,C 180,E1 -16783.35,E2 -16783.35} C_VEL
LIN {X 0,Y 321.497,Z 529.43,A -85,B 0,C 180,E1 -16785.392,E2 -16785.392} C_VEL
LIN {X 0,Y 320.619,Z 546.489,A -85,B 0,C 180,E1 -16785.869,E2 -16785.869} C_VEL
LIN {X 0,Y 319.163,Z 561.367,A -85,B 0,C 180,E1 -16786.502,E2 -16786.502} C_VEL
LIN {X 0,Y 317.236,Z 576.096,A -85,B 0,C 180,E1 -16787.384,E2 -16787.384} C_VEL
LIN {X 0,Y 314.898,Z 589.348,A -85,B 0,C 180,E1 -16788.397,E2 -16788.397} C_VEL
LIN {X 0,Y 312.225,Z 603.562,A -85,B 0,C 180,E1 -16789.814,E2 -16789.814} C_VEL
LIN {X 0,Y 309.293,Z 616.011,A -85,B 0,C 180,E1 -16791.327,E2 -16791.327} C_VEL
LIN {X 0,Y 306.136,Z 628.188,A -85,B 0,C 180,E1 -16793.148,E2 -16793.148} C_VEL
LIN {X 0,Y 303.255,Z 638.42,A -85,B 0,C 180,E1 -16794.999,E2 -16794.999} C_VEL
LIN {X 0,Y 300.468,Z 647.879,A -85,B 0,C 180,E1 -16797.056,E2 -16797.056} C_VEL
LIN {X 0,Y 297.612,Z 657.067,A -85,B 0,C 180,E1 -16799.488,E2 -16799.488} C_VEL
LIN {X 0,Y 295.598,Z 663.626,A -85,B 0,C 180,E1 -16801.607,E2 -16801.607} C_VEL
LIN {X 0,Y 293.364,Z 670.839,A -85,B 0,C 180,E1 -16804.455,E2 -16804.455} C_VEL
LIN {X 0,Y 291.703,Z 676.451,A -85,B 0,C 180,E1 -16807.326,E2 -16807.326} C_VEL
LIN {X 0,Y 290.575,Z 680.629,A -85,B 0,C 180,E1 -16810.208,E2 -16810.208} C_VEL
LIN {X 0,Y 289.828,Z 683.501,A -85,B 0,C 180,E1 -16813.083,E2 -16813.083} C_VEL
LIN {X 0,Y 289.474,Z 685.235,A -85,B 0,C 180,E1 -16816.205,E2 -16816.205} C_VEL
LIN {X 0,Y 289.293,Z 685.633,A -85,B 0,C 180,E1 -16818.793,E2 -16818.793} C_VEL
LIN {X 0,Y 289.283,Z 684.95,A -85,B 0,C 180,E1 -16821.618,E2 -16821.618} C_VEL
LIN {X 0,Y 289.56,Z 683.071,A -85,B 0,C 180,E1 -16824.429,E2 -16824.429} C_VEL
LIN {X 0,Y 289.787,Z 680.034,A -85,B 0,C 180,E1 -16827.22,E2 -16827.22} C_VEL
LIN {X 0,Y 290.324,Z 675.767,A -85,B 0,C 180,E1 -16830,E2 -16830} C_VEL
LIN {X 0,Y 291.161,Z 670.181,A -85,B 0,C 180,E1 -16832.767,E2 -16832.767} C_VEL
LIN {X 0,Y 292.48,Z 663.11,A -85,B 0,C 180,E1 -16835.516,E2 -16835.516} C_VEL
LIN {X 0,Y 294.107,Z 655.544,A -85,B 0,C 180,E1 -16837.898,E2 -16837.898} C_VEL
LIN {X 0,Y 296.001,Z 646.469,A -85,B 0,C 180,E1 -16840.258,E2 -16840.258} C_VEL
LIN {X 0,Y 297.924,Z 637.238,A -85,B 0,C 180,E1 -16842.258,E2 -16842.258} C_VEL
LIN {X 0,Y 300.471,Z 625.303,A -85,B 0,C 180,E1 -16844.39,E2 -16844.39} C_VEL
LIN {X 0,Y 302.652,Z 613.178,A -85,B 0,C 180,E1 -16846.18,E2 -16846.18} C_VEL
LIN {X 0,Y 305.01,Z 599.82,A -85,B 0,C 180,E1 -16847.777,E2 -16847.777} C_VEL
LIN {X 0,Y 306.93,Z 586.726,A -85,B 0,C 180,E1 -16849.044,E2 -16849.044} C_VEL
LIN {X 0,Y 308.75,Z 572.37,A -85,B 0,C 180,E1 -16850.138,E2 -16850.138} C_VEL
LIN {X 0,Y 310.246,Z 557.518,A -85,B 0,C 180,E1 -16850.99,E2 -16850.99} C_VEL
LIN {X 0,Y 311.274,Z 542.158,A -85,B 0,C 180,E1 -16851.611,E2 -16851.611} C_VEL
LIN {X 0,Y 312.593,Z 505.969,A -85,B 0,C 180,E1 -16852.471,E2 -16852.471} C_VEL
LIN {X 0,Y 315.305,Z 428.308,A -85,B 0,C 180,E1 -16854.204,E2 -16854.204} C_VEL
LIN {X 0,Y 312.931,Z 421.816,A -85,B 0,C 180,E1 -16854.633,E2 -16854.633} C_VEL
LIN {X 0,Y 304.812,Z 403.276,A -85,B 0,C 180,E1 -16856.066,E2 -16856.066} C_VEL
LIN {X 0,Y 298.787,Z 391.387,A -85,B 0,C 180,E1 -16857.141,E2 -16857.141} C_VEL
LIN {X 0,Y 293.051,Z 381.595,A -85,B 0,C 180,E1 -16858.172,E2 -16858.172} C_VEL
LIN {X 0,Y 291.678,Z 379.226,A -85,B 0,C 180,E1 -16858.427,E2 -16858.427} C_VEL
LIN {X 0,Y 291.365,Z 377.815,A -85,B 0,C 180,E1 -16858.538,E2 -16858.538} C_VEL
LIN {X 0,Y 291.34,Z 377.809,A -85,B 0,C 180,E1 -16862.451,E2 -16862.451} C_VEL
LIN {X 0,Y 291.359,Z 377.81,A -85,B 0,C 180,E1 -16865.374,E2 -16865.374} C_VEL
LIN {X 0,Y 291.323,Z 377.817,A -85,B 0,C 180,E1 -16868.452,E2 -16868.452} C_VEL
LIN {X 0,Y 290.681,Z 377.907,A -85,B 0,C 180,E1 -16869.606,E2 -16869.606} C_VEL
LIN {X 0,Y 287.836,Z 378.268,A -85,B 0,C 180,E1 -16871.484,E2 -16871.484} C_VEL
LIN {X 0,Y 285.393,Z 378.566,A -85,B 0,C 180,E1 -16873.009,E2 -16873.009} C_VEL
LIN {X 0,Y 284.323,Z 378.689,A -85,B 0,C 180,E1 -16874.19,E2 -16874.19} C_VEL
LIN {X 0,Y 284.225,Z 378.694,A -85,B 0,C 180,E1 -16874.591,E2 -16874.591} C_VEL
LIN {X 0,Y 284.243,Z 378.7,A -85,B 0,C 180,E1 -16878.118,E2 -16878.118} C_VEL
LIN {X 0,Y 284.284,Z 378.696,A -85,B 0,C 180,E1 -16882.288,E2 -16882.288} C_VEL
LIN {X 0,Y 284.31,Z 378.688,A -85,B 0,C 180,E1 -16885.35,E2 -16885.35} C_VEL
LIN {X 0,Y 284.288,Z 378.7,A -85,B 0,C 180,E1 -16888.724,E2 -16888.724} C_VEL
LIN {X 0,Y 284.276,Z 378.659,A -85,B 0,C 180,E1 -16891.983,E2 -16891.983} C_VEL
LIN {X 0,Y 284.295,Z 378.665,A -85,B 0,C 180,E1 -16896.159,E2 -16896.159} C_VEL
LIN {X 0,Y 284.379,Z 378.686,A -85,B 0,C 180,E1 -16899.904,E2 -16899.904} C_VEL
LIN {X 0,Y 284.457,Z 378.673,A -85,B 0,C 180,E1 -16904.486,E2 -16904.486} C_VEL
LIN {X 0,Y 284.485,Z 378.652,A -85,B 0,C 180,E1 -16908.601,E2 -16908.601} C_VEL
LIN {X 0,Y 284.611,Z 378.656,A -85,B 0,C 180,E1 -16911.479,E2 -16911.479} C_VEL
LIN {X 0,Y 284.57,Z 378.645,A -85,B 0,C 180,E1 -16914.33,E2 -16914.33} C_VEL
LIN {X 0,Y 284.847,Z 378.626,A -85,B 0,C 180,E1 -16918.586,E2 -16918.586} C_VEL
LIN {X 0,Y 284.844,Z 378.61,A -85,B 0,C 180,E1 -16921.413,E2 -16921.413} C_VEL
LIN {X 0,Y 284.644,Z 378.643,A -85,B 0,C 180,E1 -16927.091,E2 -16927.091} C_VEL
LIN {X 0,Y 284.515,Z 378.669,A -85,B 0,C 180,E1 -16929.957,E2 -16929.957} C_VEL
LIN {X 0,Y 284.435,Z 378.673,A -85,B 0,C 180,E1 -16934.305,E2 -16934.305} C_VEL
LIN {X 0,Y 284.371,Z 378.677,A -85,B 0,C 180,E1 -16938.74,E2 -16938.74} C_VEL
LIN {X 0,Y 284.324,Z 378.683,A -85,B 0,C 180,E1 -16941.763,E2 -16941.763} C_VEL
LIN {X 0,Y 284.309,Z 378.693,A -85,B 0,C 180,E1 -16944.849,E2 -16944.849} C_VEL
LIN {X 0,Y 284.283,Z 378.699,A -85,B 0,C 180,E1 -16948.015,E2 -16948.015} C_VEL
LIN {X 0,Y 284.285,Z 378.698,A -85,B 0,C 180,E1 -16951.275,E2 -16951.275} C_VEL
LIN {X 0,Y 284.336,Z 378.689,A -85,B 0,C 180,E1 -16955.346,E2 -16955.346} C_VEL
LIN {X 0,Y 284.263,Z 378.694,A -85,B 0,C 180,E1 -16958.176,E2 -16958.176} C_VEL
LIN {X 0,Y 284.236,Z 378.703,A -85,B 0,C 180,E1 -16962.117,E2 -16962.117} C_VEL
LIN {X 0,Y 284.237,Z 378.705,A -85,B 0,C 180,E1 -16966.185,E2 -16966.185} C_VEL
LIN {X 0,Y 284.239,Z 378.728,A -85,B 0,C 180,E1 -16967.195,E2 -16967.195} C_VEL
LIN {X 0,Y 287.611,Z 390.36,A -85,B 0,C 180,E1 -16970.94,E2 -16970.94} C_VEL
LIN {X 0,Y 296.13,Z 407.925,A -85,B 0,C 180,E1 -16972.589,E2 -16972.589} C_VEL
LIN {X 0,Y 305.158,Z 429,A -85,B 0,C 180,E1 -16974.275,E2 -16974.275} C_VEL
LIN {X 0,Y 306.634,Z 433.128,A -85,B 0,C 180,E1 -16974.557,E2 -16974.557} C_VEL
LIN {X 0,Y 308.723,Z 446.86,A -85,B 0,C 180,E1 -16975.162,E2 -16975.162} C_VEL
LIN {X 0,Y 304.824,Z 556.293,A -85,B 0,C 180,E1 -16977.682,E2 -16977.682} C_VEL
LIN {X 0,Y 303.603,Z 572.069,A -85,B 0,C 180,E1 -16978.27,E2 -16978.27} C_VEL
LIN {X 0,Y 301.898,Z 587.171,A -85,B 0,C 180,E1 -16979.096,E2 -16979.096} C_VEL
LIN {X 0,Y 299.774,Z 602.837,A -85,B 0,C 180,E1 -16980.271,E2 -16980.271} C_VEL
LIN {X 0,Y 297.521,Z 616.68,A -85,B 0,C 180,E1 -16981.615,E2 -16981.615} C_VEL
LIN {X 0,Y 295.011,Z 630.338,A -85,B 0,C 180,E1 -16983.278,E2 -16983.278} C_VEL
LIN {X 0,Y 292.437,Z 642.734,A -85,B 0,C 180,E1 -16985.129,E2 -16985.129} C_VEL
LIN {X 0,Y 290.144,Z 654.047,A -85,B 0,C 180,E1 -16987.197,E2 -16987.197} C_VEL
LIN {X 0,Y 288.161,Z 663.556,A -85,B 0,C 180,E1 -16989.29,E2 -16989.29} C_VEL
LIN {X 0,Y 286.168,Z 672.88,A -85,B 0,C 180,E1 -16991.752,E2 -16991.752} C_VEL
LIN {X 0,Y 284.587,Z 681.043,A -85,B 0,C 180,E1 -16994.389,E2 -16994.389} C_VEL
LIN {X 0,Y 283.516,Z 687.836,A -85,B 0,C 180,E1 -16997.109,E2 -16997.109} C_VEL
LIN {X 0,Y 282.755,Z 693.504,A -85,B 0,C 180,E1 -16999.98,E2 -16999.98} C_VEL
LIN {X 0,Y 282.464,Z 697.795,A -85,B 0,C 180,E1 -17002.853,E2 -17002.853} C_VEL
LIN {X 0,Y 282.323,Z 700.802,A -85,B 0,C 180,E1 -17005.717,E2 -17005.717} C_VEL
LIN {X 0,Y 282.354,Z 702.606,A -85,B 0,C 180,E1 -17008.574,E2 -17008.574} C_VEL
LIN {X 0,Y 282.346,Z 703.218,A -85,B 0,C 180,E1 -17011.426,E2 -17011.426} C_VEL
LIN {X 0,Y 282.288,Z 702.645,A -85,B 0,C 180,E1 -17014.283,E2 -17014.283} C_VEL
LIN {X 0,Y 282.388,Z 700.942,A -85,B 0,C 180,E1 -17017.148,E2 -17017.148} C_VEL
LIN {X 0,Y 282.832,Z 698.089,A -85,B 0,C 180,E1 -17020.017,E2 -17020.017} C_VEL
LIN {X 0,Y 283.724,Z 694.028,A -85,B 0,C 180,E1 -17022.881,E2 -17022.881} C_VEL
LIN {X 0,Y 285.046,Z 688.645,A -85,B 0,C 180,E1 -17025.736,E2 -17025.736} C_VEL
LIN {X 0,Y 287.076,Z 681.812,A -85,B 0,C 180,E1 -17028.558,E2 -17028.558} C_VEL
LIN {X 0,Y 289.626,Z 673.361,A -85,B 0,C 180,E1 -17031.345,E2 -17031.345} C_VEL
LIN {X 0,Y 292.522,Z 664.378,A -85,B 0,C 180,E1 -17033.73,E2 -17033.73} C_VEL
LIN {X 0,Y 295.217,Z 655.243,A -85,B 0,C 180,E1 -17035.751,E2 -17035.751} C_VEL
LIN {X 0,Y 298.401,Z 644.51,A -85,B 0,C 180,E1 -17037.72,E2 -17037.72} C_VEL
LIN {X 0,Y 301.703,Z 632.833,A -85,B 0,C 180,E1 -17039.478,E2 -17039.478} C_VEL
LIN {X 0,Y 304.925,Z 620.114,A -85,B 0,C 180,E1 -17041.045,E2 -17041.045} C_VEL
LIN {X 0,Y 307.876,Z 606.401,A -85,B 0,C 180,E1 -17042.413,E2 -17042.413} C_VEL
LIN {X 0,Y 310.432,Z 592.652,A -85,B 0,C 180,E1 -17043.493,E2 -17043.493} C_VEL
LIN {X 0,Y 312.736,Z 577.711,A -85,B 0,C 180,E1 -17044.376,E2 -17044.376} C_VEL
LIN {X 0,Y 314.461,Z 563.133,A -85,B 0,C 180,E1 -17044.988,E2 -17044.988} C_VEL
LIN {X 0,Y 315.558,Z 547.149,A -85,B 0,C 180,E1 -17045.431,E2 -17045.431} C_VEL
LIN {X 0,Y 319.788,Z 449.392,A -85,B 0,C 180,E1 -17047.635,E2 -17047.635} C_VEL
LIN {X 0,Y 318.894,Z 445.01,A -85,B 0,C 180,E1 -17047.905,E2 -17047.905} C_VEL
LIN {X 0,Y 311.052,Z 428.392,A -85,B 0,C 180,E1 -17049.717,E2 -17049.717} C_VEL
LIN {X 0,Y 303.583,Z 414.468,A -85,B 0,C 180,E1 -17051.528,E2 -17051.528} C_VEL
LIN {X 0,Y 296.673,Z 403.027,A -85,B 0,C 180,E1 -17053.294,E2 -17053.294} C_VEL
LIN {X 0,Y 293.994,Z 398.713,A -85,B 0,C 180,E1 -17054.014,E2 -17054.014} C_VEL
LIN {X 0,Y 290.548,Z 393.417,A -85,B 0,C 180,E1 -17054.967,E2 -17054.967} C_VEL
LIN {X 0,Y 287.723,Z 388.862,A -85,B 0,C 180,E1 -17055.832,E2 -17055.832} C_VEL
LIN {X 0,Y 285.078,Z 381.19,A -85,B 0,C 180,E1 -17059.211,E2 -17059.211} C_VEL
LIN {X 0,Y 284.303,Z 378.692,A -85,B 0,C 180,E1 -17060.387,E2 -17060.387} C_VEL
LIN {X 0,Y 284.335,Z 378.668,A -85,B 0,C 180,E1 -17064.654,E2 -17064.654} C_VEL
LIN {X 0,Y 284.285,Z 378.665,A -85,B 0,C 180,E1 -17068.725,E2 -17068.725} C_VEL
LIN {X 0,Y 284.288,Z 378.697,A -85,B 0,C 180,E1 -17071.985,E2 -17071.985} C_VEL
LIN {X 0,Y 284.324,Z 378.689,A -85,B 0,C 180,E1 -17076.146,E2 -17076.146} C_VEL
LIN {X 0,Y 284.388,Z 378.679,A -85,B 0,C 180,E1 -17079.898,E2 -17079.898} C_VEL
LIN {X 0,Y 284.493,Z 378.664,A -85,B 0,C 180,E1 -17084.46,E2 -17084.46} C_VEL
LIN {X 0,Y 284.484,Z 378.666,A -85,B 0,C 180,E1 -17088.602,E2 -17088.602} C_VEL
LIN {X 0,Y 284.609,Z 378.647,A -85,B 0,C 180,E1 -17091.48,E2 -17091.48} C_VEL
LIN {X 0,Y 284.574,Z 378.659,A -85,B 0,C 180,E1 -17094.331,E2 -17094.331} C_VEL
LIN {X 0,Y 284.845,Z 378.622,A -85,B 0,C 180,E1 -17098.587,E2 -17098.587} C_VEL
LIN {X 0,Y 284.848,Z 378.628,A -85,B 0,C 180,E1 -17101.414,E2 -17101.414} C_VEL
LIN {X 0,Y 284.644,Z 378.643,A -85,B 0,C 180,E1 -17107.092,E2 -17107.092} C_VEL
LIN {X 0,Y 284.519,Z 378.667,A -85,B 0,C 180,E1 -17109.958,E2 -17109.958} C_VEL
LIN {X 0,Y 284.484,Z 378.666,A -85,B 0,C 180,E1 -17114.303,E2 -17114.303} C_VEL
LIN {X 0,Y 284.426,Z 378.675,A -85,B 0,C 180,E1 -17117.249,E2 -17117.249} C_VEL
LIN {X 0,Y 284.378,Z 378.651,A -85,B 0,C 180,E1 -17120.243,E2 -17120.243} C_VEL
LIN {X 0,Y 284.297,Z 378.685,A -85,B 0,C 180,E1 -17123.842,E2 -17123.842} C_VEL
LIN {X 0,Y 284.291,Z 378.694,A -85,B 0,C 180,E1 -17128.016,E2 -17128.016} C_VEL
LIN {X 0,Y 284.289,Z 378.673,A -85,B 0,C 180,E1 -17131.276,E2 -17131.276} C_VEL
LIN {X 0,Y 284.312,Z 378.697,A -85,B 0,C 180,E1 -17133.448,E2 -17133.448} C_VEL
LIN {X 0,Y 285.189,Z 381.334,A -85,B 0,C 180,E1 -17133.781,E2 -17133.781} C_VEL
LIN {X 0,Y 287.13,Z 383.527,A -85,B 0,C 180,E1 -17134.336,E2 -17134.336} C_VEL
LIN {X 0,Y 287.942,Z 384.283,A -85,B 0,C 180,E1 -17134.557,E2 -17134.557} C_VEL
LIN {X 0,Y 289.975,Z 387.51,A -85,B 0,C 180,E1 -17135.152,E2 -17135.152} C_VEL
LIN {X 0,Y 291.637,Z 389.485,A -85,B 0,C 180,E1 -17135.601,E2 -17135.601} C_VEL
LIN {X 0,Y 299.319,Z 400.318,A -85,B 0,C 180,E1 -17137.625,E2 -17137.625} C_VEL
LIN {X 0,Y 307.636,Z 413.853,A -85,B 0,C 180,E1 -17139.679,E2 -17139.679} C_VEL
LIN {X 0,Y 315.08,Z 427.564,A -85,B 0,C 180,E1 -17141.415,E2 -17141.415} C_VEL
LIN {X 0,Y 320.247,Z 438.146,A -85,B 0,C 180,E1 -17142.575,E2 -17142.575} C_VEL
LIN {X 0,Y 316.012,Z 529.064,A -85,B 0,C 180,E1 -17144.581,E2 -17144.581} C_VEL
LIN {X 0,Y 315.061,Z 546.733,A -85,B 0,C 180,E1 -17145.077,E2 -17145.077} C_VEL
LIN {X 0,Y 313.563,Z 561.434,A -85,B 0,C 180,E1 -17145.708,E2 -17145.708} C_VEL
LIN {X 0,Y 311.584,Z 576.193,A -85,B 0,C 180,E1 -17146.603,E2 -17146.603} C_VEL
LIN {X 0,Y 309.086,Z 589.789,A -85,B 0,C 180,E1 -17147.653,E2 -17147.653} C_VEL
LIN {X 0,Y 306.453,Z 603.247,A -85,B 0,C 180,E1 -17149.009,E2 -17149.009} C_VEL
LIN {X 0,Y 303.252,Z 616.372,A -85,B 0,C 180,E1 -17150.622,E2 -17150.622} C_VEL
LIN {X 0,Y 299.973,Z 628.525,A -85,B 0,C 180,E1 -17152.472,E2 -17152.472} C_VEL
LIN {X 0,Y 296.691,Z 639.571,A -85,B 0,C 180,E1 -17154.524,E2 -17154.524} C_VEL
LIN {X 0,Y 293.816,Z 648.873,A -85,B 0,C 180,E1 -17156.622,E2 -17156.622} C_VEL
LIN {X 0,Y 290.869,Z 657.924,A -85,B 0,C 180,E1 -17159.106,E2 -17159.106} C_VEL
LIN {X 0,Y 288.334,Z 665.716,A -85,B 0,C 180,E1 -17161.753,E2 -17161.753} C_VEL
LIN {X 0,Y 286.189,Z 672.281,A -85,B 0,C 180,E1 -17164.548,E2 -17164.548} C_VEL
LIN {X 0,Y 284.535,Z 677.611,A -85,B 0,C 180,E1 -17167.49,E2 -17167.49} C_VEL
LIN {X 0,Y 283.428,Z 681.536,A -85,B 0,C 180,E1 -17170.438,E2 -17170.438} C_VEL
LIN {X 0,Y 282.821,Z 683.596,A -85,B 0,C 180,E1 -17172.651,E2 -17172.651} C_VEL
LIN {X 0,Y 282.414,Z 685.32,A -85,B 0,C 180,E1 -17175.59,E2 -17175.59} C_VEL
LIN {X 0,Y 282.206,Z 685.871,A -85,B 0,C 180,E1 -17178.508,E2 -17178.508} C_VEL
LIN {X 0,Y 282.195,Z 685.224,A -85,B 0,C 180,E1 -17181.406,E2 -17181.406} C_VEL
LIN {X 0,Y 282.476,Z 683.334,A -85,B 0,C 180,E1 -17184.393,E2 -17184.393} C_VEL
LIN {X 0,Y 282.695,Z 680.453,A -85,B 0,C 180,E1 -17187.15,E2 -17187.15} C_VEL
LIN {X 0,Y 283.249,Z 676.262,A -85,B 0,C 180,E1 -17190,E2 -17190} C_VEL
LIN {X 0,Y 284.103,Z 670.757,A -85,B 0,C 180,E1 -17192.836,E2 -17192.836} C_VEL
LIN {X 0,Y 285.437,Z 663.777,A -85,B 0,C 180,E1 -17195.652,E2 -17195.652} C_VEL
LIN {X 0,Y 287.109,Z 656.31,A -85,B 0,C 180,E1 -17198.091,E2 -17198.091} C_VEL
LIN {X 0,Y 289.053,Z 647.34,A -85,B 0,C 180,E1 -17200.507,E2 -17200.507} C_VEL
LIN {X 0,Y 291.392,Z 636.533,A -85,B 0,C 180,E1 -17202.891,E2 -17202.891} C_VEL
LIN {X 0,Y 293.862,Z 625.411,A -85,B 0,C 180,E1 -17204.898,E2 -17204.898} C_VEL
LIN {X 0,Y 296.135,Z 613.26,A -85,B 0,C 180,E1 -17206.724,E2 -17206.724} C_VEL
LIN {X 0,Y 298.591,Z 599.86,A -85,B 0,C 180,E1 -17208.35,E2 -17208.35} C_VEL
LIN {X 0,Y 300.582,Z 586.727,A -85,B 0,C 180,E1 -17209.64,E2 -17209.64} C_VEL
LIN {X 0,Y 302.465,Z 572.307,A -85,B 0,C 180,E1 -17210.753,E2 -17210.753} C_VEL
LIN {X 0,Y 304.002,Z 557.362,A -85,B 0,C 180,E1 -17211.62,E2 -17211.62} C_VEL
LIN {X 0,Y 305.082,Z 541.81,A -85,B 0,C 180,E1 -17212.251,E2 -17212.251} C_VEL
LIN {X 0,Y 307.385,Z 480.187,A -85,B 0,C 180,E1 -17213.693,E2 -17213.693} C_VEL
LIN {X 0,Y 309.072,Z 429.436,A -85,B 0,C 180,E1 -17214.861,E2 -17214.861} C_VEL
LIN {X 0,Y 301.692,Z 411.794,A -85,B 0,C 180,E1 -17216.207,E2 -17216.207} C_VEL
LIN {X 0,Y 294.015,Z 396.008,A -85,B 0,C 180,E1 -17217.624,E2 -17217.624} C_VEL
LIN {X 0,Y 285.9,Z 382.338,A -85,B 0,C 180,E1 -17219.137,E2 -17219.137} C_VEL
LIN {X 0,Y 284.483,Z 379.591,A -85,B 0,C 180,E1 -17219.424,E2 -17219.424} C_VEL
LIN {X 0,Y 284.322,Z 378.686,A -85,B 0,C 180,E1 -17219.508,E2 -17219.508} C_VEL
LIN {X 0,Y 284.309,Z 378.685,A -85,B 0,C 180,E1 -17222.945,E2 -17222.945} C_VEL
LIN {X 0,Y 284.325,Z 378.681,A -85,B 0,C 180,E1 -17226.387,E2 -17226.387} C_VEL
LIN {X 0,Y 284.285,Z 378.684,A -85,B 0,C 180,E1 -17229.998,E2 -17229.998} C_VEL
LIN {X 0,Y 284.25,Z 378.698,A -85,B 0,C 180,E1 -17234.19,E2 -17234.19} C_VEL
LIN {X 0,Y 284.225,Z 378.694,A -85,B 0,C 180,E1 -17234.591,E2 -17234.591} C_VEL
LIN {X 0,Y 283.532,Z 378.773,A -85,B 0,C 180,E1 -17235.774,E2 -17235.774} C_VEL
LIN {X 0,Y 280.685,Z 379.137,A -85,B 0,C 180,E1 -17237.702,E2 -17237.702} C_VEL
LIN {X 0,Y 278.291,Z 379.447,A -85,B 0,C 180,E1 -17239.267,E2 -17239.267} C_VEL
LIN {X 0,Y 277.271,Z 379.566,A -85,B 0,C 180,E1 -17240.48,E2 -17240.48} C_VEL
LIN {X 0,Y 277.19,Z 379.573,A -85,B 0,C 180,E1 -17240.891,E2 -17240.891} C_VEL
LIN {X 0,Y 277.28,Z 379.569,A -85,B 0,C 180,E1 -17244.34,E2 -17244.34} C_VEL
LIN {X 0,Y 277.243,Z 379.579,A -85,B 0,C 180,E1 -17247.835,E2 -17247.835} C_VEL
LIN {X 0,Y 277.238,Z 379.55,A -85,B 0,C 180,E1 -17251.206,E2 -17251.206} C_VEL
LIN {X 0,Y 277.234,Z 379.52,A -85,B 0,C 180,E1 -17254.471,E2 -17254.471} C_VEL
LIN {X 0,Y 277.253,Z 379.564,A -85,B 0,C 180,E1 -17257.651,E2 -17257.651} C_VEL
LIN {X 0,Y 277.327,Z 379.561,A -85,B 0,C 180,E1 -17260.764,E2 -17260.764} C_VEL
LIN {X 0,Y 277.417,Z 379.552,A -85,B 0,C 180,E1 -17265.324,E2 -17265.324} C_VEL
LIN {X 0,Y 277.46,Z 379.533,A -85,B 0,C 180,E1 -17269.786,E2 -17269.786} C_VEL
LIN {X 0,Y 277.602,Z 379.526,A -85,B 0,C 180,E1 -17272.727,E2 -17272.727} C_VEL
LIN {X 0,Y 277.813,Z 379.502,A -85,B 0,C 180,E1 -17278.55,E2 -17278.55} C_VEL
LIN {X 0,Y 277.811,Z 379.486,A -85,B 0,C 180,E1 -17281.449,E2 -17281.449} C_VEL
LIN {X 0,Y 277.602,Z 379.519,A -85,B 0,C 180,E1 -17287.272,E2 -17287.272} C_VEL
LIN {X 0,Y 277.456,Z 379.547,A -85,B 0,C 180,E1 -17290.213,E2 -17290.213} C_VEL
LIN {X 0,Y 277.387,Z 379.551,A -85,B 0,C 180,E1 -17294.676,E2 -17294.676} C_VEL
LIN {X 0,Y 277.327,Z 379.557,A -85,B 0,C 180,E1 -17299.235,E2 -17299.235} C_VEL
LIN {X 0,Y 277.286,Z 379.568,A -85,B 0,C 180,E1 -17303.924,E2 -17303.924} C_VEL
LIN {X 0,Y 277.27,Z 379.569,A -85,B 0,C 180,E1 -17307.482,E2 -17307.482} C_VEL
LIN {X 0,Y 277.248,Z 379.572,A -85,B 0,C 180,E1 -17310.472,E2 -17310.472} C_VEL
LIN {X 0,Y 277.245,Z 379.574,A -85,B 0,C 180,E1 -17313.895,E2 -17313.895} C_VEL
LIN {X 0,Y 277.232,Z 379.576,A -85,B 0,C 180,E1 -17317.474,E2 -17317.474} C_VEL
LIN {X 0,Y 277.176,Z 379.582,A -85,B 0,C 180,E1 -17321.242,E2 -17321.242} C_VEL
LIN {X 0,Y 277.173,Z 379.586,A -85,B 0,C 180,E1 -17325.232,E2 -17325.232} C_VEL
LIN {X 0,Y 277.227,Z 379.654,A -85,B 0,C 180,E1 -17326.378,E2 -17326.378} C_VEL
LIN {X 0,Y 280.284,Z 390.273,A -85,B 0,C 180,E1 -17329.885,E2 -17329.885} C_VEL
LIN {X 0,Y 287.61,Z 404.772,A -85,B 0,C 180,E1 -17331.371,E2 -17331.371} C_VEL
LIN {X 0,Y 293.556,Z 417.727,A -85,B 0,C 180,E1 -17332.54,E2 -17332.54} C_VEL
LIN {X 0,Y 300.624,Z 434.828,A -85,B 0,C 180,E1 -17333.901,E2 -17333.901} C_VEL
LIN {X 0,Y 302.613,Z 448.287,A -85,B 0,C 180,E1 -17334.506,E2 -17334.506} C_VEL
LIN {X 0,Y 298.549,Z 557.348,A -85,B 0,C 180,E1 -17337.068,E2 -17337.068} C_VEL
LIN {X 0,Y 297.217,Z 573.433,A -85,B 0,C 180,E1 -17337.707,E2 -17337.707} C_VEL
LIN {X 0,Y 295.439,Z 588.182,A -85,B 0,C 180,E1 -17338.548,E2 -17338.548} C_VEL
LIN {X 0,Y 293.313,Z 603.206,A -85,B 0,C 180,E1 -17339.718,E2 -17339.718} C_VEL
LIN {X 0,Y 290.952,Z 617.152,A -85,B 0,C 180,E1 -17341.111,E2 -17341.111} C_VEL
LIN {X 0,Y 288.569,Z 629.476,A -85,B 0,C 180,E1 -17342.632,E2 -17342.632} C_VEL
LIN {X 0,Y 285.903,Z 641.982,A -85,B 0,C 180,E1 -17344.521,E2 -17344.521} C_VEL
LIN {X 0,Y 283.481,Z 653.376,A -85,B 0,C 180,E1 -17346.63,E2 -17346.63} C_VEL
LIN {X 0,Y 281.108,Z 664.421,A -85,B 0,C 180,E1 -17349.129,E2 -17349.129} C_VEL
LIN {X 0,Y 279.107,Z 673.58,A -85,B 0,C 180,E1 -17351.654,E2 -17351.654} C_VEL
LIN {X 0,Y 277.427,Z 681.88,A -85,B 0,C 180,E1 -17354.468,E2 -17354.468} C_VEL
LIN {X 0,Y 276.28,Z 689.002,A -85,B 0,C 180,E1 -17357.513,E2 -17357.513} C_VEL
LIN {X 0,Y 275.589,Z 694.373,A -85,B 0,C 180,E1 -17360.458,E2 -17360.458} C_VEL
LIN {X 0,Y 275.37,Z 697.461,A -85,B 0,C 180,E1 -17362.668,E2 -17362.668} C_VEL
LIN {X 0,Y 275.235,Z 700.512,A -85,B 0,C 180,E1 -17365.607,E2 -17365.607} C_VEL
LIN {X 0,Y 275.278,Z 702.358,A -85,B 0,C 180,E1 -17368.537,E2 -17368.537} C_VEL
LIN {X 0,Y 275.27,Z 702.989,A -85,B 0,C 180,E1 -17371.463,E2 -17371.463} C_VEL
LIN {X 0,Y 275.203,Z 702.455,A -85,B 0,C 180,E1 -17374.394,E2 -17374.394} C_VEL
LIN {X 0,Y 275.304,Z 700.792,A -85,B 0,C 180,E1 -17377.333,E2 -17377.333} C_VEL
LIN {X 0,Y 275.788,Z 697.981,A -85,B 0,C 180,E1 -17380.276,E2 -17380.276} C_VEL
LIN {X 0,Y 276.747,Z 693.965,A -85,B 0,C 180,E1 -17383.212,E2 -17383.212} C_VEL
LIN {X 0,Y 278.247,Z 688.28,A -85,B 0,C 180,E1 -17386.301,E2 -17386.301} C_VEL
LIN {X 0,Y 280.28,Z 681.828,A -85,B 0,C 180,E1 -17389.025,E2 -17389.025} C_VEL
LIN {X 0,Y 282.986,Z 673.438,A -85,B 0,C 180,E1 -17391.872,E2 -17391.872} C_VEL
LIN {X 0,Y 285.983,Z 664.511,A -85,B 0,C 180,E1 -17394.307,E2 -17394.307} C_VEL
LIN {X 0,Y 288.817,Z 655.447,A -85,B 0,C 180,E1 -17396.365,E2 -17396.365} C_VEL
LIN {X 0,Y 292.115,Z 644.8,A -85,B 0,C 180,E1 -17398.37,E2 -17398.37} C_VEL
LIN {X 0,Y 295.562,Z 633.23,A -85,B 0,C 180,E1 -17400.154,E2 -17400.154} C_VEL
LIN {X 0,Y 298.9,Z 620.651,A -85,B 0,C 180,E1 -17401.742,E2 -17401.742} C_VEL
LIN {X 0,Y 301.907,Z 607.333,A -85,B 0,C 180,E1 -17403.112,E2 -17403.112} C_VEL
LIN {X 0,Y 304.591,Z 593.642,A -85,B 0,C 180,E1 -17404.223,E2 -17404.223} C_VEL
LIN {X 0,Y 307.022,Z 579.11,A -85,B 0,C 180,E1 -17405.109,E2 -17405.109} C_VEL
LIN {X 0,Y 308.839,Z 564.208,A -85,B 0,C 180,E1 -17405.771,E2 -17405.771} C_VEL
LIN {X 0,Y 310.013,Z 548.959,A -85,B 0,C 180,E1 -17406.214,E2 -17406.214} C_VEL
LIN {X 0,Y 314.417,Z 450.639,A -85,B 0,C 180,E1 -17408.462,E2 -17408.462} C_VEL
LIN {X 0,Y 313.747,Z 447.958,A -85,B 0,C 180,E1 -17408.654,E2 -17408.654} C_VEL
LIN {X 0,Y 306.417,Z 432.243,A -85,B 0,C 180,E1 -17410.42,E2 -17410.42} C_VEL
LIN {X 0,Y 299.4,Z 419.121,A -85,B 0,C 180,E1 -17412.184,E2 -17412.184} C_VEL
LIN {X 0,Y 292.678,Z 407.735,A -85,B 0,C 180,E1 -17413.974,E2 -17413.974} C_VEL
LIN {X 0,Y 287.072,Z 398.876,A -85,B 0,C 180,E1 -17415.56,E2 -17415.56} C_VEL
LIN {X 0,Y 283.478,Z 393.46,A -85,B 0,C 180,E1 -17416.632,E2 -17416.632} C_VEL
LIN {X 0,Y 280.334,Z 388.558,A -85,B 0,C 180,E1 -17417.643,E2 -17417.643} C_VEL
LIN {X 0,Y 277.267,Z 379.561,A -85,B 0,C 180,E1 -17422.036,E2 -17422.036} C_VEL
LIN {X 0,Y 277.245,Z 379.573,A -85,B 0,C 180,E1 -17426.105,E2 -17426.105} C_VEL
LIN {X 0,Y 277.261,Z 379.538,A -85,B 0,C 180,E1 -17429.539,E2 -17429.539} C_VEL
LIN {X 0,Y 277.295,Z 379.564,A -85,B 0,C 180,E1 -17432.858,E2 -17432.858} C_VEL
LIN {X 0,Y 277.286,Z 379.566,A -85,B 0,C 180,E1 -17436.076,E2 -17436.076} C_VEL
LIN {X 0,Y 277.343,Z 379.555,A -85,B 0,C 180,E1 -17440.767,E2 -17440.767} C_VEL
LIN {X 0,Y 277.435,Z 379.549,A -85,B 0,C 180,E1 -17445.327,E2 -17445.327} C_VEL
LIN {X 0,Y 277.458,Z 379.549,A -85,B 0,C 180,E1 -17449.788,E2 -17449.788} C_VEL
LIN {X 0,Y 277.602,Z 379.525,A -85,B 0,C 180,E1 -17452.728,E2 -17452.728} C_VEL
LIN {X 0,Y 277.692,Z 379.519,A -85,B 0,C 180,E1 -17457.099,E2 -17457.099} C_VEL
LIN {X 0,Y 277.797,Z 379.495,A -85,B 0,C 180,E1 -17460.001,E2 -17460.001} C_VEL
LIN {X 0,Y 277.654,Z 379.514,A -85,B 0,C 180,E1 -17462.902,E2 -17462.902} C_VEL
LIN {X 0,Y 277.603,Z 379.519,A -85,B 0,C 180,E1 -17467.273,E2 -17467.273} C_VEL
LIN {X 0,Y 277.462,Z 379.542,A -85,B 0,C 180,E1 -17470.214,E2 -17470.214} C_VEL
LIN {X 0,Y 277.437,Z 379.543,A -85,B 0,C 180,E1 -17474.675,E2 -17474.675} C_VEL
LIN {X 0,Y 277.344,Z 379.526,A -85,B 0,C 180,E1 -17479.235,E2 -17479.235} C_VEL
LIN {X 0,Y 277.259,Z 379.559,A -85,B 0,C 180,E1 -17483.928,E2 -17483.928} C_VEL
LIN {X 0,Y 277.274,Z 379.556,A -85,B 0,C 180,E1 -17487.484,E2 -17487.484} C_VEL
LIN {X 0,Y 277.255,Z 379.55,A -85,B 0,C 180,E1 -17491.628,E2 -17491.628} C_VEL
LIN {X 0,Y 278.107,Z 382.166,A -85,B 0,C 180,E1 -17491.999,E2 -17491.999} C_VEL
LIN {X 0,Y 280.07,Z 384.375,A -85,B 0,C 180,E1 -17492.611,E2 -17492.611} C_VEL
LIN {X 0,Y 281.026,Z 385.244,A -85,B 0,C 180,E1 -17492.893,E2 -17492.893} C_VEL
LIN {X 0,Y 283.055,Z 388.484,A -85,B 0,C 180,E1 -17493.536,E2 -17493.536} C_VEL
LIN {X 0,Y 284.814,Z 390.429,A -85,B 0,C 180,E1 -17494.045,E2 -17494.045} C_VEL
LIN {X 0,Y 287.617,Z 394.171,A -85,B 0,C 180,E1 -17494.857,E2 -17494.857} C_VEL
LIN {X 0,Y 296.124,Z 406.361,A -85,B 0,C 180,E1 -17497.177,E2 -17497.177} C_VEL
LIN {X 0,Y 304.32,Z 420.13,A -85,B 0,C 180,E1 -17499.267,E2 -17499.267} C_VEL
LIN {X 0,Y 311.521,Z 433.662,A -85,B 0,C 180,E1 -17500.997,E2 -17500.997} C_VEL
LIN {X 0,Y 314.882,Z 440.608,A -85,B 0,C 180,E1 -17501.78,E2 -17501.78} C_VEL
LIN {X 0,Y 310.423,Z 531.882,A -85,B 0,C 180,E1 -17503.809,E2 -17503.809} C_VEL
LIN {X 0,Y 309.539,Z 547.627,A -85,B 0,C 180,E1 -17504.282,E2 -17504.282} C_VEL
LIN {X 0,Y 307.977,Z 562.097,A -85,B 0,C 180,E1 -17504.917,E2 -17504.917} C_VEL
LIN {X 0,Y 306.11,Z 575.506,A -85,B 0,C 180,E1 -17505.735,E2 -17505.735} C_VEL
LIN {X 0,Y 303.332,Z 590.261,A -85,B 0,C 180,E1 -17506.882,E2 -17506.882} C_VEL
LIN {X 0,Y 300.738,Z 602.971,A -85,B 0,C 180,E1 -17508.176,E2 -17508.176} C_VEL
LIN {X 0,Y 297.61,Z 615.543,A -85,B 0,C 180,E1 -17509.725,E2 -17509.725} C_VEL
LIN {X 0,Y 294.452,Z 626.863,A -85,B 0,C 180,E1 -17511.424,E2 -17511.424} C_VEL
LIN {X 0,Y 291.261,Z 637.366,A -85,B 0,C 180,E1 -17513.33,E2 -17513.33} C_VEL
LIN {X 0,Y 288.162,Z 647.01,A -85,B 0,C 180,E1 -17515.456,E2 -17515.456} C_VEL
LIN {X 0,Y 284.993,Z 656.428,A -85,B 0,C 180,E1 -17517.981,E2 -17517.981} C_VEL
LIN {X 0,Y 282.145,Z 664.54,A -85,B 0,C 180,E1 -17520.673,E2 -17520.673} C_VEL
LIN {X 0,Y 280.056,Z 670.549,A -85,B 0,C 180,E1 -17523.147,E2 -17523.147} C_VEL
LIN {X 0,Y 278.117,Z 676.331,A -85,B 0,C 180,E1 -17526.152,E2 -17526.152} C_VEL
LIN {X 0,Y 276.744,Z 680.669,A -85,B 0,C 180,E1 -17529.174,E2 -17529.174} C_VEL
LIN {X 0,Y 275.842,Z 683.692,A -85,B 0,C 180,E1 -17532.197,E2 -17532.197} C_VEL
LIN {X 0,Y 275.343,Z 685.489,A -85,B 0,C 180,E1 -17535.212,E2 -17535.212} C_VEL
LIN {X 0,Y 275.134,Z 686.09,A -85,B 0,C 180,E1 -17538.209,E2 -17538.209} C_VEL
LIN {X 0,Y 275.089,Z 685.499,A -85,B 0,C 180,E1 -17541.183,E2 -17541.183} C_VEL
LIN {X 0,Y 275.401,Z 683.547,A -85,B 0,C 180,E1 -17544.42,E2 -17544.42} C_VEL
LIN {X 0,Y 275.604,Z 680.871,A -85,B 0,C 180,E1 -17547.077,E2 -17547.077} C_VEL
LIN {X 0,Y 276.175,Z 676.755,A -85,B 0,C 180,E1 -17550,E2 -17550} C_VEL
LIN {X 0,Y 277.048,Z 671.33,A -85,B 0,C 180,E1 -17552.908,E2 -17552.908} C_VEL
LIN {X 0,Y 278.395,Z 664.44,A -85,B 0,C 180,E1 -17555.796,E2 -17555.796} C_VEL
LIN {X 0,Y 280.117,Z 657.048,A -85,B 0,C 180,E1 -17558.295,E2 -17558.295} C_VEL
LIN {X 0,Y 282.113,Z 648.157,A -85,B 0,C 180,E1 -17560.769,E2 -17560.769} C_VEL
LIN {X 0,Y 284.523,Z 637.493,A -85,B 0,C 180,E1 -17563.208,E2 -17563.208} C_VEL
LIN {X 0,Y 287.262,Z 625.506,A -85,B 0,C 180,E1 -17565.43,E2 -17565.43} C_VEL
LIN {X 0,Y 289.653,Z 613.327,A -85,B 0,C 180,E1 -17567.291,E2 -17567.291} C_VEL
LIN {X 0,Y 292.2,Z 599.889,A -85,B 0,C 180,E1 -17568.948,E2 -17568.948} C_VEL
LIN {X 0,Y 294.266,Z 586.725,A -85,B 0,C 180,E1 -17570.262,E2 -17570.262} C_VEL
LIN {X 0,Y 296.19,Z 572.252,A -85,B 0,C 180,E1 -17571.397,E2 -17571.397} C_VEL
LIN {X 0,Y 297.793,Z 557.208,A -85,B 0,C 180,E1 -17572.277,E2 -17572.277} C_VEL
LIN {X 0,Y 298.917,Z 541.463,A -85,B 0,C 180,E1 -17572.918,E2 -17572.918} C_VEL
LIN {X 0,Y 303.057,Z 431.963,A -85,B 0,C 180,E1 -17575.486,E2 -17575.486} C_VEL
LIN {X 0,Y 298.633,Z 420.66,A -85,B 0,C 180,E1 -17576.333,E2 -17576.333} C_VEL
LIN {X 0,Y 290.334,Z 402.692,A -85,B 0,C 180,E1 -17577.917,E2 -17577.917} C_VEL
LIN {X 0,Y 281.284,Z 387.109,A -85,B 0,C 180,E1 -17579.659,E2 -17579.659} C_VEL
LIN {X 0,Y 279.022,Z 383.439,A -85,B 0,C 180,E1 -17580.112,E2 -17580.112} C_VEL
LIN {X 0,Y 277.521,Z 380.847,A -85,B 0,C 180,E1 -17580.422,E2 -17580.422} C_VEL
LIN {X 0,Y 277.253,Z 379.57,A -85,B 0,C 180,E1 -17580.557,E2 -17580.557} C_VEL
LIN {X 0,Y 277.25,Z 379.572,A -85,B 0,C 180,E1 -17583.896,E2 -17583.896} C_VEL
LIN {X 0,Y 277.258,Z 379.568,A -85,B 0,C 180,E1 -17587.471,E2 -17587.471} C_VEL
LIN {X 0,Y 277.188,Z 379.566,A -85,B 0,C 180,E1 -17591.241,E2 -17591.241} C_VEL
LIN {X 0,Y 277.198,Z 379.563,A -85,B 0,C 180,E1 -17595.227,E2 -17595.227} C_VEL
LIN {X 0,Y 277.18,Z 379.582,A -85,B 0,C 180,E1 -17598.757,E2 -17598.757} C_VEL
LIN {X 0,Y 277.19,Z 379.573,A -85,B 0,C 180,E1 -17600.891,E2 -17600.891} C_VEL
LIN {X 0,Y 276.541,Z 379.659,A -85,B 0,C 180,E1 -17602.105,E2 -17602.105} C_VEL
LIN {X 0,Y 273.733,Z 380.012,A -85,B 0,C 180,E1 -17604.084,E2 -17604.084} C_VEL
LIN {X 0,Y 271.328,Z 380.31,A -85,B 0,C 180,E1 -17605.691,E2 -17605.691} C_VEL
LIN {X 0,Y 270.271,Z 380.439,A -85,B 0,C 180,E1 -17606.936,E2 -17606.936} C_VEL
LIN {X 0,Y 270.172,Z 380.45,A -85,B 0,C 180,E1 -17607.358,E2 -17607.358} C_VEL
LIN {X 0,Y 270.184,Z 380.443,A -85,B 0,C 180,E1 -17610.38,E2 -17610.38} C_VEL
LIN {X 0,Y 270.182,Z 380.395,A -85,B 0,C 180,E1 -17613.754,E2 -17613.754} C_VEL
LIN {X 0,Y 270.186,Z 380.438,A -85,B 0,C 180,E1 -17617.034,E2 -17617.034} C_VEL
LIN {X 0,Y 270.263,Z 380.442,A -85,B 0,C 180,E1 -17620.241,E2 -17620.241} C_VEL
LIN {X 0,Y 270.376,Z 380.427,A -85,B 0,C 180,E1 -17624.933,E2 -17624.933} C_VEL
LIN {X 0,Y 270.412,Z 380.408,A -85,B 0,C 180,E1 -17629.517,E2 -17629.517} C_VEL
LIN {X 0,Y 270.564,Z 380.403,A -85,B 0,C 180,E1 -17632.537,E2 -17632.537} C_VEL
LIN {X 0,Y 270.778,Z 380.378,A -85,B 0,C 180,E1 -17638.512,E2 -17638.512} C_VEL
LIN {X 0,Y 270.776,Z 380.362,A -85,B 0,C 180,E1 -17641.487,E2 -17641.487} C_VEL
LIN {X 0,Y 270.564,Z 380.394,A -85,B 0,C 180,E1 -17647.462,E2 -17647.462} C_VEL
LIN {X 0,Y 270.407,Z 380.424,A -85,B 0,C 180,E1 -17650.482,E2 -17650.482} C_VEL
LIN {X 0,Y 270.352,Z 380.428,A -85,B 0,C 180,E1 -17655.067,E2 -17655.067} C_VEL
LIN {X 0,Y 270.293,Z 380.437,A -85,B 0,C 180,E1 -17659.756,E2 -17659.756} C_VEL
LIN {X 0,Y 270.225,Z 380.447,A -85,B 0,C 180,E1 -17664.59,E2 -17664.59} C_VEL
LIN {X 0,Y 270.2,Z 380.454,A -85,B 0,C 180,E1 -17667.916,E2 -17667.916} C_VEL
LIN {X 0,Y 270.173,Z 380.457,A -85,B 0,C 180,E1 -17671.349,E2 -17671.349} C_VEL
LIN {X 0,Y 270.197,Z 380.453,A -85,B 0,C 180,E1 -17674.906,E2 -17674.906} C_VEL
LIN {X 0,Y 270.167,Z 380.443,A -85,B 0,C 180,E1 -17678.702,E2 -17678.702} C_VEL
LIN {X 0,Y 270.147,Z 380.459,A -85,B 0,C 180,E1 -17683.245,E2 -17683.245} C_VEL
LIN {X 0,Y 270.175,Z 380.646,A -85,B 0,C 180,E1 -17685.523,E2 -17685.523} C_VEL
LIN {X 0,Y 272.905,Z 389.942,A -85,B 0,C 180,E1 -17688.745,E2 -17688.745} C_VEL
LIN {X 0,Y 280.263,Z 404.082,A -85,B 0,C 180,E1 -17690.311,E2 -17690.311} C_VEL
LIN {X 0,Y 287.57,Z 419.758,A -85,B 0,C 180,E1 -17691.811,E2 -17691.811} C_VEL
LIN {X 0,Y 294.887,Z 437.507,A -85,B 0,C 180,E1 -17693.276,E2 -17693.276} C_VEL
LIN {X 0,Y 296.549,Z 448.836,A -85,B 0,C 180,E1 -17693.801,E2 -17693.801} C_VEL
LIN {X 0,Y 292.387,Z 557.004,A -85,B 0,C 180,E1 -17696.386,E2 -17696.386} C_VEL
LIN {X 0,Y 291.001,Z 573.134,A -85,B 0,C 180,E1 -17697.033,E2 -17697.033} C_VEL
LIN {X 0,Y 289.157,Z 588.078,A -85,B 0,C 180,E1 -17697.902,E2 -17697.902} C_VEL
LIN {X 0,Y 287.014,Z 602.693,A -85,B 0,C 180,E1 -17699.055,E2 -17699.055} C_VEL
LIN {X 0,Y 284.693,Z 616.17,A -85,B 0,C 180,E1 -17700.414,E2 -17700.414} C_VEL
LIN {X 0,Y 281.93,Z 629.834,A -85,B 0,C 180,E1 -17702.134,E2 -17702.134} C_VEL
LIN {X 0,Y 279.192,Z 642.243,A -85,B 0,C 180,E1 -17704.063,E2 -17704.063} C_VEL
LIN {X 0,Y 276.603,Z 653.921,A -85,B 0,C 180,E1 -17706.297,E2 -17706.297} C_VEL
LIN {X 0,Y 274.406,Z 663.833,A -85,B 0,C 180,E1 -17708.594,E2 -17708.594} C_VEL
LIN {X 0,Y 272.25,Z 673.042,A -85,B 0,C 180,E1 -17711.175,E2 -17711.175} C_VEL
LIN {X 0,Y 270.535,Z 681.205,A -85,B 0,C 180,E1 -17713.984,E2 -17713.984} C_VEL
LIN {X 0,Y 269.522,Z 686.976,A -85,B 0,C 180,E1 -17716.427,E2 -17716.427} C_VEL
LIN {X 0,Y 268.662,Z 692.744,A -85,B 0,C 180,E1 -17719.449,E2 -17719.449} C_VEL
LIN {X 0,Y 268.294,Z 697.126,A -85,B 0,C 180,E1 -17722.474,E2 -17722.474} C_VEL
LIN {X 0,Y 268.151,Z 700.221,A -85,B 0,C 180,E1 -17725.49,E2 -17725.49} C_VEL
LIN {X 0,Y 268.203,Z 702.104,A -85,B 0,C 180,E1 -17728.498,E2 -17728.498} C_VEL
LIN {X 0,Y 268.194,Z 702.76,A -85,B 0,C 180,E1 -17731.502,E2 -17731.502} C_VEL
LIN {X 0,Y 268.107,Z 702.266,A -85,B 0,C 180,E1 -17734.51,E2 -17734.51} C_VEL
LIN {X 0,Y 268.241,Z 700.645,A -85,B 0,C 180,E1 -17737.527,E2 -17737.527} C_VEL
LIN {X 0,Y 268.76,Z 697.877,A -85,B 0,C 180,E1 -17740.547,E2 -17740.547} C_VEL
LIN {X 0,Y 269.787,Z 693.896,A -85,B 0,C 180,E1 -17743.559,E2 -17743.559} C_VEL
LIN {X 0,Y 271.282,Z 688.579,A -85,B 0,C 180,E1 -17746.557,E2 -17746.557} C_VEL
LIN {X 0,Y 273.529,Z 681.844,A -85,B 0,C 180,E1 -17749.513,E2 -17749.513} C_VEL
LIN {X 0,Y 276.384,Z 673.509,A -85,B 0,C 180,E1 -17752.422,E2 -17752.422} C_VEL
LIN {X 0,Y 279.314,Z 665.167,A -85,B 0,C 180,E1 -17754.774,E2 -17754.774} C_VEL
LIN {X 0,Y 282.448,Z 655.663,A -85,B 0,C 180,E1 -17757.007,E2 -17757.007} C_VEL
LIN {X 0,Y 285.874,Z 645.107,A -85,B 0,C 180,E1 -17759.048,E2 -17759.048} C_VEL
LIN {X 0,Y 289.454,Z 633.644,A -85,B 0,C 180,E1 -17760.859,E2 -17760.859} C_VEL
LIN {X 0,Y 292.916,Z 621.2,A -85,B 0,C 180,E1 -17762.469,E2 -17762.469} C_VEL
LIN {X 0,Y 296.135,Z 607.604,A -85,B 0,C 180,E1 -17763.897,E2 -17763.897} C_VEL
LIN {X 0,Y 299.005,Z 593.515,A -85,B 0,C 180,E1 -17765.057,E2 -17765.057} C_VEL
LIN {X 0,Y 301.462,Z 579.025,A -85,B 0,C 180,E1 -17765.958,E2 -17765.958} C_VEL
LIN {X 0,Y 303.497,Z 563.069,A -85,B 0,C 180,E1 -17766.656,E2 -17766.656} C_VEL
LIN {X 0,Y 304.65,Z 547.273,A -85,B 0,C 180,E1 -17767.113,E2 -17767.113} C_VEL
LIN {X 0,Y 309.137,Z 452.047,A -85,B 0,C 180,E1 -17769.309,E2 -17769.309} C_VEL
LIN {X 0,Y 302.168,Z 436.83,A -85,B 0,C 180,E1 -17771.056,E2 -17771.056} C_VEL
LIN {X 0,Y 295.254,Z 423.723,A -85,B 0,C 180,E1 -17772.863,E2 -17772.863} C_VEL
LIN {X 0,Y 287.406,Z 410.133,A -85,B 0,C 180,E1 -17775.059,E2 -17775.059} C_VEL
LIN {X 0,Y 282.733,Z 403.013,A -85,B 0,C 180,E1 -17776.439,E2 -17776.439} C_VEL
LIN {X 0,Y 279.907,Z 398.672,A -85,B 0,C 180,E1 -17777.319,E2 -17777.319} C_VEL
LIN {X 0,Y 276.319,Z 393.351,A -85,B 0,C 180,E1 -17778.482,E2 -17778.482} C_VEL
LIN {X 0,Y 273.013,Z 388.495,A -85,B 0,C 180,E1 -17779.61,E2 -17779.61} C_VEL
LIN {X 0,Y 270.944,Z 382.805,A -85,B 0,C 180,E1 -17782.443,E2 -17782.443} C_VEL
LIN {X 0,Y 270.218,Z 380.422,A -85,B 0,C 180,E1 -17783.733,E2 -17783.733} C_VEL
LIN {X 0,Y 270.2,Z 380.444,A -85,B 0,C 180,E1 -17786.893,E2 -17786.893} C_VEL
LIN {X 0,Y 270.184,Z 380.426,A -85,B 0,C 180,E1 -17790.382,E2 -17790.382} C_VEL
LIN {X 0,Y 270.207,Z 380.443,A -85,B 0,C 180,E1 -17793.759,E2 -17793.759} C_VEL
LIN {X 0,Y 270.207,Z 380.443,A -85,B 0,C 180,E1 -17797.037,E2 -17797.037} C_VEL
LIN {X 0,Y 270.301,Z 380.432,A -85,B 0,C 180,E1 -17800.245,E2 -17800.245} C_VEL
LIN {X 0,Y 270.404,Z 380.421,A -85,B 0,C 180,E1 -17804.936,E2 -17804.936} C_VEL
LIN {X 0,Y 270.411,Z 380.426,A -85,B 0,C 180,E1 -17809.518,E2 -17809.518} C_VEL
LIN {X 0,Y 270.564,Z 380.399,A -85,B 0,C 180,E1 -17812.538,E2 -17812.538} C_VEL
LIN {X 0,Y 270.779,Z 380.375,A -85,B 0,C 180,E1 -17818.513,E2 -17818.513} C_VEL
LIN {X 0,Y 270.778,Z 380.381,A -85,B 0,C 180,E1 -17821.488,E2 -17821.488} C_VEL
LIN {X 0,Y 270.564,Z 380.396,A -85,B 0,C 180,E1 -17827.463,E2 -17827.463} C_VEL
LIN {X 0,Y 270.414,Z 380.418,A -85,B 0,C 180,E1 -17830.483,E2 -17830.483} C_VEL
LIN {X 0,Y 270.405,Z 380.419,A -85,B 0,C 180,E1 -17835.065,E2 -17835.065} C_VEL
LIN {X 0,Y 270.291,Z 380.403,A -85,B 0,C 180,E1 -17839.757,E2 -17839.757} C_VEL
LIN {X 0,Y 270.18,Z 380.429,A -85,B 0,C 180,E1 -17844.596,E2 -17844.596} C_VEL
LIN {X 0,Y 270.204,Z 380.444,A -85,B 0,C 180,E1 -17847.917,E2 -17847.917} C_VEL
LIN {X 0,Y 270.218,Z 380.568,A -85,B 0,C 180,E1 -17849.685,E2 -17849.685} C_VEL
LIN {X 0,Y 271.098,Z 383.119,A -85,B 0,C 180,E1 -17850.063,E2 -17850.063} C_VEL
LIN {X 0,Y 273.284,Z 385.444,A -85,B 0,C 180,E1 -17850.802,E2 -17850.802} C_VEL
LIN {X 0,Y 274.102,Z 386.152,A -85,B 0,C 180,E1 -17851.066,E2 -17851.066} C_VEL
LIN {X 0,Y 276.14,Z 389.411,A -85,B 0,C 180,E1 -17851.771,E2 -17851.771} C_VEL
LIN {X 0,Y 278.011,Z 391.345,A -85,B 0,C 180,E1 -17852.356,E2 -17852.356} C_VEL
LIN {X 0,Y 280.524,Z 394.895,A -85,B 0,C 180,E1 -17853.155,E2 -17853.155} C_VEL
LIN {X 0,Y 281.806,Z 396.529,A -85,B 0,C 180,E1 -17853.544,E2 -17853.544} C_VEL
LIN {X 0,Y 285.655,Z 401.836,A -85,B 0,C 180,E1 -17854.687,E2 -17854.687} C_VEL
LIN {X 0,Y 292.5,Z 411.672,A -85,B 0,C 180,E1 -17856.598,E2 -17856.598} C_VEL
LIN {X 0,Y 300.928,Z 426.13,A -85,B 0,C 180,E1 -17858.82,E2 -17858.82} C_VEL
LIN {X 0,Y 308.181,Z 440.23,A -85,B 0,C 180,E1 -17860.62,E2 -17860.62} C_VEL
LIN {X 0,Y 309.47,Z 442.944,A -85,B 0,C 180,E1 -17860.932,E2 -17860.932} C_VEL
LIN {X 0,Y 306.39,Z 506.985,A -85,B 0,C 180,E1 -17862.402,E2 -17862.402} C_VEL
LIN {X 0,Y 304.644,Z 540.439,A -85,B 0,C 180,E1 -17863.179,E2 -17863.179} C_VEL
LIN {X 0,Y 303.344,Z 555.345,A -85,B 0,C 180,E1 -17863.733,E2 -17863.733} C_VEL
LIN {X 0,Y 301.579,Z 569.039,A -85,B 0,C 180,E1 -17864.458,E2 -17864.458} C_VEL
LIN {X 0,Y 299.032,Z 584.067,A -85,B 0,C 180,E1 -17865.519,E2 -17865.519} C_VEL
LIN {X 0,Y 296.542,Z 595.963,A -85,B 0,C 180,E1 -17866.584,E2 -17866.584} C_VEL
LIN {X 0,Y 293.438,Z 609.482,A -85,B 0,C 180,E1 -17868.116,E2 -17868.116} C_VEL
LIN {X 0,Y 290.014,Z 621.811,A -85,B 0,C 180,E1 -17869.818,E2 -17869.818} C_VEL
LIN {X 0,Y 286.567,Z 632.99,A -85,B 0,C 180,E1 -17871.703,E2 -17871.703} C_VEL
LIN {X 0,Y 283.118,Z 643.52,A -85,B 0,C 180,E1 -17873.874,E2 -17873.874} C_VEL
LIN {X 0,Y 279.63,Z 653.576,A -85,B 0,C 180,E1 -17876.432,E2 -17876.432} C_VEL
LIN {X 0,Y 276.606,Z 661.892,A -85,B 0,C 180,E1 -17879.035,E2 -17879.035} C_VEL
LIN {X 0,Y 274.124,Z 668.725,A -85,B 0,C 180,E1 -17881.686,E2 -17881.686} C_VEL
LIN {X 0,Y 271.797,Z 675.123,A -85,B 0,C 180,E1 -17884.827,E2 -17884.827} C_VEL
LIN {X 0,Y 270.191,Z 679.731,A -85,B 0,C 180,E1 -17887.842,E2 -17887.842} C_VEL
LIN {X 0,Y 269.33,Z 682.399,A -85,B 0,C 180,E1 -17890.17,E2 -17890.17} C_VEL
LIN {X 0,Y 268.524,Z 684.874,A -85,B 0,C 180,E1 -17893.268,E2 -17893.268} C_VEL
LIN {X 0,Y 268.206,Z 686.124,A -85,B 0,C 180,E1 -17896.359,E2 -17896.359} C_VEL
LIN {X 0,Y 267.957,Z 686.178,A -85,B 0,C 180,E1 -17899.421,E2 -17899.421} C_VEL
LIN {X 0,Y 268.072,Z 685.084,A -85,B 0,C 180,E1 -17902.468,E2 -17902.468} C_VEL
LIN {X 0,Y 268.353,Z 682.843,A -85,B 0,C 180,E1 -17905.494,E2 -17905.494} C_VEL
LIN {X 0,Y 268.725,Z 679.424,A -85,B 0,C 180,E1 -17908.501,E2 -17908.501} C_VEL
LIN {X 0,Y 269.452,Z 674.745,A -85,B 0,C 180,E1 -17911.495,E2 -17911.495} C_VEL
LIN {X 0,Y 270.587,Z 668.692,A -85,B 0,C 180,E1 -17914.469,E2 -17914.469} C_VEL
LIN {X 0,Y 272.304,Z 661.076,A -85,B 0,C 180,E1 -17917.415,E2 -17917.415} C_VEL
LIN {X 0,Y 274.262,Z 652.944,A -85,B 0,C 180,E1 -17919.961,E2 -17919.961} C_VEL
LIN {X 0,Y 276.539,Z 643.201,A -85,B 0,C 180,E1 -17922.475,E2 -17922.475} C_VEL
LIN {X 0,Y 278.897,Z 633.222,A -85,B 0,C 180,E1 -17924.596,E2 -17924.596} C_VEL
LIN {X 0,Y 281.576,Z 621.373,A -85,B 0,C 180,E1 -17926.681,E2 -17926.681} C_VEL
LIN {X 0,Y 283.99,Z 609.56,A -85,B 0,C 180,E1 -17928.393,E2 -17928.393} C_VEL
LIN {X 0,Y 286.352,Z 596.796,A -85,B 0,C 180,E1 -17929.91,E2 -17929.91} C_VEL
LIN {X 0,Y 288.558,Z 582.837,A -85,B 0,C 180,E1 -17931.241,E2 -17931.241} C_VEL
LIN {X 0,Y 290.369,Z 568.409,A -85,B 0,C 180,E1 -17932.315,E2 -17932.315} C_VEL
LIN {X 0,Y 291.985,Z 552.594,A -85,B 0,C 180,E1 -17933.166,E2 -17933.166} C_VEL
LIN {X 0,Y 292.962,Z 536.638,A -85,B 0,C 180,E1 -17933.739,E2 -17933.739} C_VEL
LIN {X 0,Y 296.984,Z 433.915,A -85,B 0,C 180,E1 -17936.162,E2 -17936.162} C_VEL
LIN {X 0,Y 294.207,Z 426.503,A -85,B 0,C 180,E1 -17936.72,E2 -17936.72} C_VEL
LIN {X 0,Y 286.623,Z 409.599,A -85,B 0,C 180,E1 -17938.215,E2 -17938.215} C_VEL
LIN {X 0,Y 282.16,Z 401.184,A -85,B 0,C 180,E1 -17939.097,E2 -17939.097} C_VEL
LIN {X 0,Y 274.033,Z 387.612,A -85,B 0,C 180,E1 -17940.748,E2 -17940.748} C_VEL
LIN {X 0,Y 271.934,Z 384.284,A -85,B 0,C 180,E1 -17941.191,E2 -17941.191} C_VEL
LIN {X 0,Y 270.472,Z 381.619,A -85,B 0,C 180,E1 -17941.516,E2 -17941.516} C_VEL
LIN {X 0,Y 270.206,Z 380.447,A -85,B 0,C 180,E1 -17941.622,E2 -17941.622} C_VEL
LIN {X 0,Y 270.202,Z 380.45,A -85,B 0,C 180,E1 -17944.906,E2 -17944.906} C_VEL
LIN {X 0,Y 270.201,Z 380.453,A -85,B 0,C 180,E1 -17948.71,E2 -17948.71} C_VEL
LIN {X 0,Y 270.161,Z 380.459,A -85,B 0,C 180,E1 -17953.247,E2 -17953.247} C_VEL
LIN {X 0,Y 270.154,Z 380.446,A -85,B 0,C 180,E1 -17957.437,E2 -17957.437} C_VEL
LIN {X 0,Y 270.154,Z 380.449,A -85,B 0,C 180,E1 -17961.364,E2 -17961.364} C_VEL
LIN {X 0,Y 270.2,Z 380.446,A -85,B 0,C 180,E1 -17965.093,E2 -17965.093} C_VEL
LIN {X 0,Y 270.172,Z 380.45,A -85,B 0,C 180,E1 -17967.358,E2 -17967.358} C_VEL
LIN {X 0,Y 269.465,Z 380.548,A -85,B 0,C 180,E1 -17968.603,E2 -17968.603} C_VEL
LIN {X 0,Y 266.592,Z 380.884,A -85,B 0,C 180,E1 -17970.633,E2 -17970.633} C_VEL
LIN {X 0,Y 264.183,Z 381.156,A -85,B 0,C 180,E1 -17972.282,E2 -17972.282} C_VEL
LIN {X 0,Y 263.161,Z 381.269,A -85,B 0,C 180,E1 -17973.561,E2 -17973.561} C_VEL
LIN {X 0,Y 263.083,Z 381.278,A -85,B 0,C 180,E1 -17973.994,E2 -17973.994} C_VEL
LIN {X 0,Y 263.133,Z 381.327,A -85,B 0,C 180,E1 -17978.041,E2 -17978.041} C_VEL
LIN {X 0,Y 263.223,Z 381.309,A -85,B 0,C 180,E1 -17981.312,E2 -17981.312} C_VEL
LIN {X 0,Y 263.317,Z 381.306,A -85,B 0,C 180,E1 -17984.519,E2 -17984.519} C_VEL
LIN {X 0,Y 263.352,Z 381.285,A -85,B 0,C 180,E1 -17989.233,E2 -17989.233} C_VEL
LIN {X 0,Y 263.528,Z 381.28,A -85,B 0,C 180,E1 -17992.336,E2 -17992.336} C_VEL
LIN {X 0,Y 263.741,Z 381.255,A -85,B 0,C 180,E1 -17998.472,E2 -17998.472} C_VEL
LIN {X 0,Y 263.74,Z 381.237,A -85,B 0,C 180,E1 -18001.526,E2 -18001.526} C_VEL
LIN {X 0,Y 263.528,Z 381.27,A -85,B 0,C 180,E1 -18007.662,E2 -18007.662} C_VEL
LIN {X 0,Y 263.345,Z 381.304,A -85,B 0,C 180,E1 -18010.766,E2 -18010.766} C_VEL
LIN {X 0,Y 263.299,Z 381.31,A -85,B 0,C 180,E1 -18015.48,E2 -18015.48} C_VEL
LIN {X 0,Y 263.261,Z 381.313,A -85,B 0,C 180,E1 -18020.306,E2 -18020.306} C_VEL
LIN {X 0,Y 263.168,Z 381.324,A -85,B 0,C 180,E1 -18025.295,E2 -18025.295} C_VEL
LIN {X 0,Y 263.134,Z 381.332,A -85,B 0,C 180,E1 -18028.734,E2 -18028.734} C_VEL
LIN {X 0,Y 263.128,Z 381.331,A -85,B 0,C 180,E1 -18032.288,E2 -18032.288} C_VEL
LIN {X 0,Y 263.153,Z 381.326,A -85,B 0,C 180,E1 -18035.983,E2 -18035.983} C_VEL
LIN {X 0,Y 263.071,Z 381.324,A -85,B 0,C 180,E1 -18039.878,E2 -18039.878} C_VEL
LIN {X 0,Y 263.086,Z 381.338,A -85,B 0,C 180,E1 -18044.391,E2 -18044.391} C_VEL
LIN {X 0,Y 263.086,Z 381.378,A -85,B 0,C 180,E1 -18044.525,E2 -18044.525} C_VEL
LIN {X 0,Y 265.565,Z 389.752,A -85,B 0,C 180,E1 -18047.534,E2 -18047.534} C_VEL
LIN {X 0,Y 274.947,Z 407.397,A -85,B 0,C 180,E1 -18049.623,E2 -18049.623} C_VEL
LIN {X 0,Y 282.811,Z 424.532,A -85,B 0,C 180,E1 -18051.302,E2 -18051.302} C_VEL
LIN {X 0,Y 289.163,Z 440.218,A -85,B 0,C 180,E1 -18052.625,E2 -18052.625} C_VEL
LIN {X 0,Y 290.528,Z 450.202,A -85,B 0,C 180,E1 -18053.092,E2 -18053.092} C_VEL
LIN {X 0,Y 286.256,Z 556.557,A -85,B 0,C 180,E1 -18055.673,E2 -18055.673} C_VEL
LIN {X 0,Y 284.921,Z 571.983,A -85,B 0,C 180,E1 -18056.289,E2 -18056.289} C_VEL
LIN {X 0,Y 282.987,Z 587.546,A -85,B 0,C 180,E1 -18057.2,E2 -18057.2} C_VEL
LIN {X 0,Y 280.729,Z 602.402,A -85,B 0,C 180,E1 -18058.387,E2 -18058.387} C_VEL
LIN {X 0,Y 278.158,Z 616.629,A -85,B 0,C 180,E1 -18059.856,E2 -18059.856} C_VEL
LIN {X 0,Y 275.319,Z 630.174,A -85,B 0,C 180,E1 -18061.612,E2 -18061.612} C_VEL
LIN {X 0,Y 272.5,Z 642.494,A -85,B 0,C 180,E1 -18063.583,E2 -18063.583} C_VEL
LIN {X 0,Y 269.804,Z 654.135,A -85,B 0,C 180,E1 -18065.876,E2 -18065.876} C_VEL
LIN {X 0,Y 267.371,Z 664.637,A -85,B 0,C 180,E1 -18068.408,E2 -18068.408} C_VEL
LIN {X 0,Y 265.184,Z 673.682,A -85,B 0,C 180,E1 -18071.055,E2 -18071.055} C_VEL
LIN {X 0,Y 263.513,Z 681.275,A -85,B 0,C 180,E1 -18073.765,E2 -18073.765} C_VEL
LIN {X 0,Y 262.271,Z 688.176,A -85,B 0,C 180,E1 -18076.834,E2 -18076.834} C_VEL
LIN {X 0,Y 261.498,Z 693.624,A -85,B 0,C 180,E1 -18079.939,E2 -18079.939} C_VEL
LIN {X 0,Y 261.217,Z 696.788,A -85,B 0,C 180,E1 -18082.269,E2 -18082.269} C_VEL
LIN {X 0,Y 261.064,Z 699.929,A -85,B 0,C 180,E1 -18085.368,E2 -18085.368} C_VEL
LIN {X 0,Y 261.13,Z 701.842,A -85,B 0,C 180,E1 -18088.458,E2 -18088.458} C_VEL
LIN {X 0,Y 261.12,Z 702.531,A -85,B 0,C 180,E1 -18091.542,E2 -18091.542} C_VEL
LIN {X 0,Y 261.051,Z 701.939,A -85,B 0,C 180,E1 -18095.059,E2 -18095.059} C_VEL
LIN {X 0,Y 261.174,Z 700.498,A -85,B 0,C 180,E1 -18097.732,E2 -18097.732} C_VEL
LIN {X 0,Y 261.726,Z 697.773,A -85,B 0,C 180,E1 -18100.834,E2 -18100.834} C_VEL
LIN {X 0,Y 262.837,Z 693.817,A -85,B 0,C 180,E1 -18103.925,E2 -18103.925} C_VEL
LIN {X 0,Y 264.415,Z 688.546,A -85,B 0,C 180,E1 -18107,E2 -18107} C_VEL
LIN {X 0,Y 266.782,Z 681.865,A -85,B 0,C 180,E1 -18110.027,E2 -18110.027} C_VEL
LIN {X 0,Y 269.356,Z 674.705,A -85,B 0,C 180,E1 -18112.635,E2 -18112.635} C_VEL
LIN {X 0,Y 272.431,Z 666.571,A -85,B 0,C 180,E1 -18115.063,E2 -18115.063} C_VEL
LIN {X 0,Y 275.59,Z 657.502,A -85,B 0,C 180,E1 -18117.325,E2 -18117.325} C_VEL
LIN {X 0,Y 279.108,Z 647.321,A -85,B 0,C 180,E1 -18119.407,E2 -18119.407} C_VEL
LIN {X 0,Y 282.999,Z 635.2,A -85,B 0,C 180,E1 -18121.434,E2 -18121.434} C_VEL
LIN {X 0,Y 286.968,Z 621.811,A -85,B 0,C 180,E1 -18123.218,E2 -18123.218} C_VEL
LIN {X 0,Y 290.306,Z 608.322,A -85,B 0,C 180,E1 -18124.673,E2 -18124.673} C_VEL
LIN {X 0,Y 293.277,Z 594.453,A -85,B 0,C 180,E1 -18125.846,E2 -18125.846} C_VEL
LIN {X 0,Y 296.019,Z 578.94,A -85,B 0,C 180,E1 -18126.833,E2 -18126.833} C_VEL
LIN {X 0,Y 298.116,Z 563.069,A -85,B 0,C 180,E1 -18127.536,E2 -18127.536} C_VEL
LIN {X 0,Y 299.313,Z 547.368,A -85,B 0,C 180,E1 -18127.998,E2 -18127.998} C_VEL
LIN {X 0,Y 303.838,Z 454.321,A -85,B 0,C 180,E1 -18130.176,E2 -18130.176} C_VEL
LIN {X 0,Y 297.52,Z 440.533,A -85,B 0,C 180,E1 -18131.827,E2 -18131.827} C_VEL
LIN {X 0,Y 291.263,Z 428.452,A -85,B 0,C 180,E1 -18133.534,E2 -18133.534} C_VEL
LIN {X 0,Y 283.487,Z 414.918,A -85,B 0,C 180,E1 -18135.793,E2 -18135.793} C_VEL
LIN {X 0,Y 276.864,Z 404.502,A -85,B 0,C 180,E1 -18137.87,E2 -18137.87} C_VEL
LIN {X 0,Y 272.955,Z 398.69,A -85,B 0,C 180,E1 -18139.182,E2 -18139.182} C_VEL
LIN {X 0,Y 268.972,Z 393.005,A -85,B 0,C 180,E1 -18140.593,E2 -18140.593} C_VEL
LIN {X 0,Y 265.731,Z 388.287,A -85,B 0,C 180,E1 -18141.815,E2 -18141.815} C_VEL
LIN {X 0,Y 265.412,Z 387.696,A -85,B 0,C 180,E1 -18142.002,E2 -18142.002} C_VEL
LIN {X 0,Y 263.156,Z 381.317,A -85,B 0,C 180,E1 -18145.655,E2 -18145.655} C_VEL
LIN {X 0,Y 263.125,Z 381.298,A -85,B 0,C 180,E1 -18149.504,E2 -18149.504} C_VEL
LIN {X 0,Y 263.144,Z 381.325,A -85,B 0,C 180,E1 -18152.998,E2 -18152.998} C_VEL
LIN {X 0,Y 263.149,Z 381.324,A -85,B 0,C 180,E1 -18156.384,E2 -18156.384} C_VEL
LIN {X 0,Y 263.263,Z 381.311,A -85,B 0,C 180,E1 -18159.694,E2 -18159.694} C_VEL
LIN {X 0,Y 263.351,Z 381.296,A -85,B 0,C 180,E1 -18164.523,E2 -18164.523} C_VEL
LIN {X 0,Y 263.351,Z 381.304,A -85,B 0,C 180,E1 -18169.234,E2 -18169.234} C_VEL
LIN {X 0,Y 263.527,Z 381.274,A -85,B 0,C 180,E1 -18172.338,E2 -18172.338} C_VEL
LIN {X 0,Y 263.744,Z 381.251,A -85,B 0,C 180,E1 -18178.474,E2 -18178.474} C_VEL
LIN {X 0,Y 263.742,Z 381.258,A -85,B 0,C 180,E1 -18181.528,E2 -18181.528} C_VEL
LIN {X 0,Y 263.528,Z 381.273,A -85,B 0,C 180,E1 -18187.664,E2 -18187.664} C_VEL
LIN {X 0,Y 263.357,Z 381.295,A -85,B 0,C 180,E1 -18190.767,E2 -18190.767} C_VEL
LIN {X 0,Y 263.353,Z 381.299,A -85,B 0,C 180,E1 -18195.479,E2 -18195.479} C_VEL
LIN {X 0,Y 263.251,Z 381.281,A -85,B 0,C 180,E1 -18200.308,E2 -18200.308} C_VEL
LIN {X 0,Y 263.129,Z 381.301,A -85,B 0,C 180,E1 -18205.3,E2 -18205.3} C_VEL
LIN {X 0,Y 263.188,Z 381.366,A -85,B 0,C 180,E1 -18207.487,E2 -18207.487} C_VEL
LIN {X 0,Y 264.004,Z 383.898,A -85,B 0,C 180,E1 -18207.883,E2 -18207.883} C_VEL
LIN {X 0,Y 265.946,Z 386.122,A -85,B 0,C 180,E1 -18208.62,E2 -18208.62} C_VEL
LIN {X 0,Y 267.211,Z 387.065,A -85,B 0,C 180,E1 -18209.063,E2 -18209.063} C_VEL
LIN {X 0,Y 269.178,Z 390.224,A -85,B 0,C 180,E1 -18209.811,E2 -18209.811} C_VEL
LIN {X 0,Y 271.271,Z 392.394,A -85,B 0,C 180,E1 -18210.528,E2 -18210.528} C_VEL
LIN {X 0,Y 273.761,Z 395.889,A -85,B 0,C 180,E1 -18211.391,E2 -18211.391} C_VEL
LIN {X 0,Y 275.145,Z 397.575,A -85,B 0,C 180,E1 -18211.846,E2 -18211.846} C_VEL
LIN {X 0,Y 281.875,Z 406.711,A -85,B 0,C 180,E1 -18213.964,E2 -18213.964} C_VEL
LIN {X 0,Y 289.129,Z 417.336,A -85,B 0,C 180,E1 -18216.066,E2 -18216.066} C_VEL
LIN {X 0,Y 297.398,Z 431.903,A -85,B 0,C 180,E1 -18218.323,E2 -18218.323} C_VEL
LIN {X 0,Y 304.261,Z 445.584,A -85,B 0,C 180,E1 -18220.087,E2 -18220.087} C_VEL
LIN {X 0,Y 299.915,Z 528.952,A -85,B 0,C 180,E1 -18221.989,E2 -18221.989} C_VEL
LIN {X 0,Y 298.803,Z 547.049,A -85,B 0,C 180,E1 -18222.505,E2 -18222.505} C_VEL
LIN {X 0,Y 297.096,Z 562.232,A -85,B 0,C 180,E1 -18223.174,E2 -18223.174} C_VEL
LIN {X 0,Y 294.937,Z 576.766,A -85,B 0,C 180,E1 -18224.089,E2 -18224.089} C_VEL
LIN {X 0,Y 291.999,Z 591.211,A -85,B 0,C 180,E1 -18225.251,E2 -18225.251} C_VEL
LIN {X 0,Y 289.07,Z 604.229,A -85,B 0,C 180,E1 -18226.62,E2 -18226.62} C_VEL
LIN {X 0,Y 285.457,Z 617.518,A -85,B 0,C 180,E1 -18228.337,E2 -18228.337} C_VEL
LIN {X 0,Y 281.638,Z 629.878,A -85,B 0,C 180,E1 -18230.319,E2 -18230.319} C_VEL
LIN {X 0,Y 278.337,Z 639.719,A -85,B 0,C 180,E1 -18232.243,E2 -18232.243} C_VEL
LIN {X 0,Y 274.651,Z 650.113,A -85,B 0,C 180,E1 -18234.726,E2 -18234.726} C_VEL
LIN {X 0,Y 271.614,Z 658.229,A -85,B 0,C 180,E1 -18237.086,E2 -18237.086} C_VEL
LIN {X 0,Y 268.828,Z 665.405,A -85,B 0,C 180,E1 -18239.626,E2 -18239.626} C_VEL
LIN {X 0,Y 266.292,Z 671.912,A -85,B 0,C 180,E1 -18242.493,E2 -18242.493} C_VEL
LIN {X 0,Y 264.163,Z 677.477,A -85,B 0,C 180,E1 -18245.646,E2 -18245.646} C_VEL
LIN {X 0,Y 263,Z 680.714,A -85,B 0,C 180,E1 -18248.03,E2 -18248.03} C_VEL
LIN {X 0,Y 261.909,Z 683.887,A -85,B 0,C 180,E1 -18251.216,E2 -18251.216} C_VEL
LIN {X 0,Y 261.25,Z 685.8,A -85,B 0,C 180,E1 -18254.394,E2 -18254.394} C_VEL
LIN {X 0,Y 260.992,Z 686.498,A -85,B 0,C 180,E1 -18257.56,E2 -18257.56} C_VEL
LIN {X 0,Y 260.882,Z 686.047,A -85,B 0,C 180,E1 -18260.698,E2 -18260.698} C_VEL
LIN {X 0,Y 261.127,Z 684.45,A -85,B 0,C 180,E1 -18263.82,E2 -18263.82} C_VEL
LIN {X 0,Y 261.426,Z 681.699,A -85,B 0,C 180,E1 -18266.918,E2 -18266.918} C_VEL
LIN {X 0,Y 262.012,Z 677.732,A -85,B 0,C 180,E1 -18270,E2 -18270} C_VEL
LIN {X 0,Y 262.927,Z 672.446,A -85,B 0,C 180,E1 -18273.065,E2 -18273.065} C_VEL
LIN {X 0,Y 264.321,Z 665.721,A -85,B 0,C 180,E1 -18276.105,E2 -18276.105} C_VEL
LIN {X 0,Y 266.385,Z 657.349,A -85,B 0,C 180,E1 -18279.108,E2 -18279.108} C_VEL
LIN {X 0,Y 268.604,Z 648.428,A -85,B 0,C 180,E1 -18281.7,E2 -18281.7} C_VEL
LIN {X 0,Y 271.234,Z 637.723,A -85,B 0,C 180,E1 -18284.25,E2 -18284.25} C_VEL
LIN {X 0,Y 274.133,Z 625.684,A -85,B 0,C 180,E1 -18286.572,E2 -18286.572} C_VEL
LIN {X 0,Y 276.786,Z 613.439,A -85,B 0,C 180,E1 -18288.506,E2 -18288.506} C_VEL
LIN {X 0,Y 279.503,Z 599.918,A -85,B 0,C 180,E1 -18290.227,E2 -18290.227} C_VEL
LIN {X 0,Y 281.726,Z 586.687,A -85,B 0,C 180,E1 -18291.59,E2 -18291.59} C_VEL
LIN {X 0,Y 283.759,Z 572.084,A -85,B 0,C 180,E1 -18292.768,E2 -18292.768} C_VEL
LIN {X 0,Y 285.501,Z 556.788,A -85,B 0,C 180,E1 -18293.676,E2 -18293.676} C_VEL
LIN {X 0,Y 286.623,Z 541.804,A -85,B 0,C 180,E1 -18294.298,E2 -18294.298} C_VEL
LIN {X 0,Y 290.97,Z 435.627,A -85,B 0,C 180,E1 -18296.87,E2 -18296.87} C_VEL
LIN {X 0,Y 284.967,Z 420.991,A -85,B 0,C 180,E1 -18298.101,E2 -18298.101} C_VEL
LIN {X 0,Y 278.719,Z 408.025,A -85,B 0,C 180,E1 -18299.387,E2 -18299.387} C_VEL
LIN {X 0,Y 269.784,Z 392.791,A -85,B 0,C 180,E1 -18301.259,E2 -18301.259} C_VEL
LIN {X 0,Y 265.68,Z 386.032,A -85,B 0,C 180,E1 -18302.166,E2 -18302.166} C_VEL
LIN {X 0,Y 263.687,Z 383.238,A -85,B 0,C 180,E1 -18302.604,E2 -18302.604} C_VEL
LIN {X 0,Y 263.159,Z 381.319,A -85,B 0,C 180,E1 -18302.796,E2 -18302.796} C_VEL
LIN {X 0,Y 263.179,Z 381.315,A -85,B 0,C 180,E1 -18306.761,E2 -18306.761} C_VEL
LIN {X 0,Y 263.095,Z 381.323,A -85,B 0,C 180,E1 -18309.875,E2 -18309.875} C_VEL
LIN {X 0,Y 263.105,Z 381.333,A -85,B 0,C 180,E1 -18313.988,E2 -18313.988} C_VEL
LIN {X 0,Y 263.077,Z 381.339,A -85,B 0,C 180,E1 -18318.418,E2 -18318.418} C_VEL
LIN {X 0,Y 263.106,Z 381.33,A -85,B 0,C 180,E1 -18322.093,E2 -18322.093} C_VEL
LIN {X 0,Y 263.154,Z 381.32,A -85,B 0,C 180,E1 -18325.885,E2 -18325.885} C_VEL
LIN {X 0,Y 263.128,Z 381.331,A -85,B 0,C 180,E1 -18329.503,E2 -18329.503} C_VEL
LIN {X 0,Y 263.117,Z 381.277,A -85,B 0,C 180,E1 -18332.993,E2 -18332.993} C_VEL
LIN {X 0,Y 263.083,Z 381.278,A -85,B 0,C 180,E1 -18333.994,E2 -18333.994} C_VEL
LIN {X 0,Y 262.449,Z 381.368,A -85,B 0,C 180,E1 -18335.272,E2 -18335.272} C_VEL
LIN {X 0,Y 259.683,Z 381.749,A -85,B 0,C 180,E1 -18337.357,E2 -18337.357} C_VEL
LIN {X 0,Y 257.306,Z 382.063,A -85,B 0,C 180,E1 -18339.052,E2 -18339.052} C_VEL
LIN {X 0,Y 256.259,Z 382.189,A -85,B 0,C 180,E1 -18340.364,E2 -18340.364} C_VEL
LIN {X 0,Y 256.16,Z 382.195,A -85,B 0,C 180,E1 -18340.809,E2 -18340.809} C_VEL
LIN {X 0,Y 256.251,Z 382.182,A -85,B 0,C 180,E1 -18344.081,E2 -18344.081} C_VEL
LIN {X 0,Y 256.293,Z 382.162,A -85,B 0,C 180,E1 -18348.933,E2 -18348.933} C_VEL
LIN {X 0,Y 256.492,Z 382.157,A -85,B 0,C 180,E1 -18352.125,E2 -18352.125} C_VEL
LIN {X 0,Y 256.454,Z 382.157,A -85,B 0,C 180,E1 -18356.857,E2 -18356.857} C_VEL
LIN {X 0,Y 256.702,Z 382.132,A -85,B 0,C 180,E1 -18358.43,E2 -18358.43} C_VEL
LIN {X 0,Y 256.703,Z 382.114,A -85,B 0,C 180,E1 -18361.568,E2 -18361.568} C_VEL
LIN {X 0,Y 256.458,Z 382.159,A -85,B 0,C 180,E1 -18366.293,E2 -18366.293} C_VEL
LIN {X 0,Y 256.428,Z 382.162,A -85,B 0,C 180,E1 -18369.464,E2 -18369.464} C_VEL
LIN {X 0,Y 256.217,Z 382.185,A -85,B 0,C 180,E1 -18374.292,E2 -18374.292} C_VEL
LIN {X 0,Y 256.175,Z 382.185,A -85,B 0,C 180,E1 -18377.564,E2 -18377.564} C_VEL
LIN {X 0,Y 256.155,Z 382.196,A -85,B 0,C 180,E1 -18381.117,E2 -18381.117} C_VEL
LIN {X 0,Y 256.134,Z 382.202,A -85,B 0,C 180,E1 -18385.111,E2 -18385.111} C_VEL
LIN {X 0,Y 256.055,Z 382.209,A -85,B 0,C 180,E1 -18389.606,E2 -18389.606} C_VEL
LIN {X 0,Y 256.066,Z 382.208,A -85,B 0,C 180,E1 -18393.292,E2 -18393.292} C_VEL
LIN {X 0,Y 256.085,Z 382.212,A -85,B 0,C 180,E1 -18397.262,E2 -18397.262} C_VEL
LIN {X 0,Y 256.009,Z 382.218,A -85,B 0,C 180,E1 -18401.212,E2 -18401.212} C_VEL
LIN {X 0,Y 256.021,Z 382.294,A -85,B 0,C 180,E1 -18403.523,E2 -18403.523} C_VEL
LIN {X 0,Y 258.158,Z 389.315,A -85,B 0,C 180,E1 -18406.216,E2 -18406.216} C_VEL
LIN {X 0,Y 268.407,Z 408.301,A -85,B 0,C 180,E1 -18408.626,E2 -18408.626} C_VEL
LIN {X 0,Y 276.267,Z 425.183,A -85,B 0,C 180,E1 -18410.383,E2 -18410.383} C_VEL
LIN {X 0,Y 283.305,Z 442.406,A -85,B 0,C 180,E1 -18411.91,E2 -18411.91} C_VEL
LIN {X 0,Y 284.547,Z 451.035,A -85,B 0,C 180,E1 -18412.336,E2 -18412.336} C_VEL
LIN {X 0,Y 280.183,Z 556.094,A -85,B 0,C 180,E1 -18414.93,E2 -18414.93} C_VEL
LIN {X 0,Y 278.814,Z 571.614,A -85,B 0,C 180,E1 -18415.557,E2 -18415.557} C_VEL
LIN {X 0,Y 276.799,Z 587.218,A -85,B 0,C 180,E1 -18416.479,E2 -18416.479} C_VEL
LIN {X 0,Y 274.598,Z 601.45,A -85,B 0,C 180,E1 -18417.628,E2 -18417.628} C_VEL
LIN {X 0,Y 271.961,Z 615.612,A -85,B 0,C 180,E1 -18419.095,E2 -18419.095} C_VEL
LIN {X 0,Y 268.959,Z 629.299,A -85,B 0,C 180,E1 -18420.877,E2 -18420.877} C_VEL
LIN {X 0,Y 266.061,Z 641.733,A -85,B 0,C 180,E1 -18422.892,E2 -18422.892} C_VEL
LIN {X 0,Y 263.357,Z 653.038,A -85,B 0,C 180,E1 -18425.138,E2 -18425.138} C_VEL
LIN {X 0,Y 260.673,Z 664.047,A -85,B 0,C 180,E1 -18427.824,E2 -18427.824} C_VEL
LIN {X 0,Y 258.375,Z 673.159,A -85,B 0,C 180,E1 -18430.536,E2 -18430.536} C_VEL
LIN {X 0,Y 256.5,Z 681.32,A -85,B 0,C 180,E1 -18433.532,E2 -18433.532} C_VEL
LIN {X 0,Y 255.285,Z 687.747,A -85,B 0,C 180,E1 -18436.467,E2 -18436.467} C_VEL
LIN {X 0,Y 254.444,Z 693.239,A -85,B 0,C 180,E1 -18439.657,E2 -18439.657} C_VEL
LIN {X 0,Y 254.139,Z 696.45,A -85,B 0,C 180,E1 -18442.052,E2 -18442.052} C_VEL
LIN {X 0,Y 253.991,Z 699.636,A -85,B 0,C 180,E1 -18445.238,E2 -18445.238} C_VEL
LIN {X 0,Y 254.057,Z 701.572,A -85,B 0,C 180,E1 -18448.415,E2 -18448.415} C_VEL
LIN {X 0,Y 254.047,Z 702.302,A -85,B 0,C 180,E1 -18451.585,E2 -18451.585} C_VEL
LIN {X 0,Y 253.943,Z 701.838,A -85,B 0,C 180,E1 -18454.923,E2 -18454.923} C_VEL
LIN {X 0,Y 254.108,Z 700.351,A -85,B 0,C 180,E1 -18457.949,E2 -18457.949} C_VEL
LIN {X 0,Y 254.689,Z 697.668,A -85,B 0,C 180,E1 -18461.137,E2 -18461.137} C_VEL
LIN {X 0,Y 255.879,Z 693.739,A -85,B 0,C 180,E1 -18464.312,E2 -18464.312} C_VEL
LIN {X 0,Y 257.59,Z 688.518,A -85,B 0,C 180,E1 -18467.465,E2 -18467.465} C_VEL
LIN {X 0,Y 260.07,Z 681.89,A -85,B 0,C 180,E1 -18470.567,E2 -18470.567} C_VEL
LIN {X 0,Y 262.789,Z 674.787,A -85,B 0,C 180,E1 -18473.233,E2 -18473.233} C_VEL
LIN {X 0,Y 265.81,Z 667.174,A -85,B 0,C 180,E1 -18475.59,E2 -18475.59} C_VEL
LIN {X 0,Y 269.283,Z 657.718,A -85,B 0,C 180,E1 -18478.02,E2 -18478.02} C_VEL
LIN {X 0,Y 272.935,Z 647.584,A -85,B 0,C 180,E1 -18480.14,E2 -18480.14} C_VEL
LIN {X 0,Y 276.988,Z 635.566,A -85,B 0,C 180,E1 -18482.197,E2 -18482.197} C_VEL
LIN {X 0,Y 281.038,Z 622.463,A -85,B 0,C 180,E1 -18483.991,E2 -18483.991} C_VEL
LIN {X 0,Y 284.126,Z 610.53,A -85,B 0,C 180,E1 -18485.328,E2 -18485.328} C_VEL
LIN {X 0,Y 287.376,Z 596.322,A -85,B 0,C 180,E1 -18486.592,E2 -18486.592} C_VEL
LIN {X 0,Y 290.006,Z 582.768,A -85,B 0,C 180,E1 -18487.509,E2 -18487.509} C_VEL
LIN {X 0,Y 292.231,Z 567.753,A -85,B 0,C 180,E1 -18488.263,E2 -18488.263} C_VEL
LIN {X 0,Y 293.781,Z 552.097,A -85,B 0,C 180,E1 -18488.79,E2 -18488.79} C_VEL
LIN {X 0,Y 298.646,Z 456.827,A -85,B 0,C 180,E1 -18491.06,E2 -18491.06} C_VEL
LIN {X 0,Y 292.692,Z 443.735,A -85,B 0,C 180,E1 -18492.69,E2 -18492.69} C_VEL
LIN {X 0,Y 286.466,Z 431.734,A -85,B 0,C 180,E1 -18494.466,E2 -18494.466} C_VEL
LIN {X 0,Y 279.574,Z 419.584,A -85,B 0,C 180,E1 -18496.564,E2 -18496.564} C_VEL
LIN {X 0,Y 273.12,Z 409.323,A -85,B 0,C 180,E1 -18498.678,E2 -18498.678} C_VEL
LIN {X 0,Y 269.636,Z 404.054,A -85,B 0,C 180,E1 -18499.898,E2 -18499.898} C_VEL
LIN {X 0,Y 265.854,Z 398.545,A -85,B 0,C 180,E1 -18501.292,E2 -18501.292} C_VEL
LIN {X 0,Y 262.086,Z 393.142,A -85,B 0,C 180,E1 -18502.77,E2 -18502.77} C_VEL
LIN {X 0,Y 258.154,Z 387.767,A -85,B 0,C 180,E1 -18504.416,E2 -18504.416} C_VEL
LIN {X 0,Y 257.317,Z 385.376,A -85,B 0,C 180,E1 -18505.72,E2 -18505.72} C_VEL
LIN {X 0,Y 256.091,Z 382.181,A -85,B 0,C 180,E1 -18507.905,E2 -18507.905} C_VEL
LIN {X 0,Y 256.095,Z 382.21,A -85,B 0,C 180,E1 -18512.191,E2 -18512.191} C_VEL
LIN {X 0,Y 256.135,Z 382.204,A -85,B 0,C 180,E1 -18515.697,E2 -18515.697} C_VEL
LIN {X 0,Y 256.164,Z 382.201,A -85,B 0,C 180,E1 -18519.105,E2 -18519.105} C_VEL
LIN {X 0,Y 256.3,Z 382.174,A -85,B 0,C 180,E1 -18524.086,E2 -18524.086} C_VEL
LIN {X 0,Y 256.292,Z 382.179,A -85,B 0,C 180,E1 -18528.934,E2 -18528.934} C_VEL
LIN {X 0,Y 256.469,Z 382.152,A -85,B 0,C 180,E1 -18532.126,E2 -18532.126} C_VEL
LIN {X 0,Y 256.489,Z 382.155,A -85,B 0,C 180,E1 -18536.859,E2 -18536.859} C_VEL
LIN {X 0,Y 256.708,Z 382.128,A -85,B 0,C 180,E1 -18538.432,E2 -18538.432} C_VEL
LIN {X 0,Y 256.703,Z 382.135,A -85,B 0,C 180,E1 -18541.57,E2 -18541.57} C_VEL
LIN {X 0,Y 256.444,Z 382.157,A -85,B 0,C 180,E1 -18546.631,E2 -18546.631} C_VEL
LIN {X 0,Y 256.429,Z 382.169,A -85,B 0,C 180,E1 -18549.466,E2 -18549.466} C_VEL
LIN {X 0,Y 256.257,Z 382.181,A -85,B 0,C 180,E1 -18554.291,E2 -18554.291} C_VEL
LIN {X 0,Y 256.211,Z 382.178,A -85,B 0,C 180,E1 -18557.563,E2 -18557.563} C_VEL
LIN {X 0,Y 256.144,Z 382.173,A -85,B 0,C 180,E1 -18561.111,E2 -18561.111} C_VEL
LIN {X 0,Y 256.106,Z 382.246,A -85,B 0,C 180,E1 -18564.99,E2 -18564.99} C_VEL
LIN {X 0,Y 256.851,Z 384.585,A -85,B 0,C 180,E1 -18565.4,E2 -18565.4} C_VEL
LIN {X 0,Y 258.481,Z 386.67,A -85,B 0,C 180,E1 -18566.113,E2 -18566.113} C_VEL
LIN {X 0,Y 260.415,Z 388.094,A -85,B 0,C 180,E1 -18566.876,E2 -18566.876} C_VEL
LIN {X 0,Y 262.316,Z 391.284,A -85,B 0,C 180,E1 -18567.684,E2 -18567.684} C_VEL
LIN {X 0,Y 264.554,Z 393.47,A -85,B 0,C 180,E1 -18568.525,E2 -18568.525} C_VEL
LIN {X 0,Y 267.142,Z 396.993,A -85,B 0,C 180,E1 -18569.503,E2 -18569.503} C_VEL
LIN {X 0,Y 268.591,Z 398.747,A -85,B 0,C 180,E1 -18570.023,E2 -18570.023} C_VEL
LIN {X 0,Y 272.852,Z 404.478,A -85,B 0,C 180,E1 -18571.508,E2 -18571.508} C_VEL
LIN {X 0,Y 278.641,Z 412.348,A -85,B 0,C 180,E1 -18573.379,E2 -18573.379} C_VEL
LIN {X 0,Y 285.702,Z 422.996,A -85,B 0,C 180,E1 -18575.502,E2 -18575.502} C_VEL
LIN {X 0,Y 293.366,Z 436.661,A -85,B 0,C 180,E1 -18577.668,E2 -18577.668} C_VEL
LIN {X 0,Y 299.097,Z 448.171,A -85,B 0,C 180,E1 -18579.205,E2 -18579.205} C_VEL
LIN {X 0,Y 294.52,Z 532.182,A -85,B 0,C 180,E1 -18581.135,E2 -18581.135} C_VEL
LIN {X 0,Y 293.422,Z 548.605,A -85,B 0,C 180,E1 -18581.637,E2 -18581.637} C_VEL
LIN {X 0,Y 291.61,Z 563.851,A -85,B 0,C 180,E1 -18582.343,E2 -18582.343} C_VEL
LIN {X 0,Y 289.194,Z 578.84,A -85,B 0,C 180,E1 -18583.319,E2 -18583.319} C_VEL
LIN {X 0,Y 286.427,Z 591.716,A -85,B 0,C 180,E1 -18584.387,E2 -18584.387} C_VEL
LIN {X 0,Y 283.386,Z 604.676,A -85,B 0,C 180,E1 -18585.773,E2 -18585.773} C_VEL
LIN {X 0,Y 279.63,Z 617.917,A -85,B 0,C 180,E1 -18587.51,E2 -18587.51} C_VEL
LIN {X 0,Y 275.782,Z 629.942,A -85,B 0,C 180,E1 -18589.471,E2 -18589.471} C_VEL
LIN {X 0,Y 271.919,Z 640.888,A -85,B 0,C 180,E1 -18591.662,E2 -18591.662} C_VEL
LIN {X 0,Y 268.386,Z 650.388,A -85,B 0,C 180,E1 -18593.993,E2 -18593.993} C_VEL
LIN {X 0,Y 264.943,Z 659.096,A -85,B 0,C 180,E1 -18596.604,E2 -18596.604} C_VEL
LIN {X 0,Y 261.922,Z 666.522,A -85,B 0,C 180,E1 -18599.348,E2 -18599.348} C_VEL
LIN {X 0,Y 259.102,Z 673.344,A -85,B 0,C 180,E1 -18602.541,E2 -18602.541} C_VEL
LIN {X 0,Y 256.97,Z 678.629,A -85,B 0,C 180,E1 -18605.78,E2 -18605.78} C_VEL
LIN {X 0,Y 255.437,Z 682.751,A -85,B 0,C 180,E1 -18609.306,E2 -18609.306} C_VEL
LIN {X 0,Y 254.522,Z 685.108,A -85,B 0,C 180,E1 -18612.318,E2 -18612.318} C_VEL
LIN {X 0,Y 254.072,Z 686.464,A -85,B 0,C 180,E1 -18615.584,E2 -18615.584} C_VEL
LIN {X 0,Y 253.788,Z 686.656,A -85,B 0,C 180,E1 -18618.823,E2 -18618.823} C_VEL
LIN {X 0,Y 253.876,Z 685.7,A -85,B 0,C 180,E1 -18622.044,E2 -18622.044} C_VEL
LIN {X 0,Y 254.16,Z 683.6,A -85,B 0,C 180,E1 -18625.242,E2 -18625.242} C_VEL
LIN {X 0,Y 254.518,Z 680.322,A -85,B 0,C 180,E1 -18628.418,E2 -18628.418} C_VEL
LIN {X 0,Y 255.3,Z 675.756,A -85,B 0,C 180,E1 -18631.578,E2 -18631.578} C_VEL
LIN {X 0,Y 256.501,Z 669.839,A -85,B 0,C 180,E1 -18634.715,E2 -18634.715} C_VEL
LIN {X 0,Y 258.281,Z 662.407,A -85,B 0,C 180,E1 -18637.82,E2 -18637.82} C_VEL
LIN {X 0,Y 260.365,Z 654.442,A -85,B 0,C 180,E1 -18640.498,E2 -18640.498} C_VEL
LIN {X 0,Y 262.787,Z 644.912,A -85,B 0,C 180,E1 -18643.14,E2 -18643.14} C_VEL
LIN {X 0,Y 265.267,Z 635.187,A -85,B 0,C 180,E1 -18645.364,E2 -18645.364} C_VEL
LIN {X 0,Y 268.125,Z 623.635,A -85,B 0,C 180,E1 -18647.544,E2 -18647.544} C_VEL
LIN {X 0,Y 270.917,Z 610.925,A -85,B 0,C 180,E1 -18649.512,E2 -18649.512} C_VEL
LIN {X 0,Y 273.458,Z 598.358,A -85,B 0,C 180,E1 -18651.088,E2 -18651.088} C_VEL
LIN {X 0,Y 275.821,Z 584.68,A -85,B 0,C 180,E1 -18652.47,E2 -18652.47} C_VEL
LIN {X 0,Y 277.771,Z 570.676,A -85,B 0,C 180,E1 -18653.583,E2 -18653.583} C_VEL
LIN {X 0,Y 279.494,Z 555.602,A -85,B 0,C 180,E1 -18654.464,E2 -18654.464} C_VEL
LIN {X 0,Y 280.579,Z 541.266,A -85,B 0,C 180,E1 -18655.054,E2 -18655.054} C_VEL
LIN {X 0,Y 284.984,Z 438.01,A -85,B 0,C 180,E1 -18657.589,E2 -18657.589} C_VEL
LIN {X 0,Y 284.494,Z 436.081,A -85,B 0,C 180,E1 -18657.713,E2 -18657.713} C_VEL
LIN {X 0,Y 277.433,Z 419.609,A -85,B 0,C 180,E1 -18659.214,E2 -18659.214} C_VEL
LIN {X 0,Y 272.833,Z 410.469,A -85,B 0,C 180,E1 -18660.198,E2 -18660.198} C_VEL
LIN {X 0,Y 264.58,Z 396.487,A -85,B 0,C 180,E1 -18661.998,E2 -18661.998} C_VEL
LIN {X 0,Y 260.174,Z 389.604,A -85,B 0,C 180,E1 -18663.003,E2 -18663.003} C_VEL
LIN {X 0,Y 258.336,Z 386.531,A -85,B 0,C 180,E1 -18663.444,E2 -18663.444} C_VEL
LIN {X 0,Y 256.68,Z 384.243,A -85,B 0,C 180,E1 -18663.832,E2 -18663.832} C_VEL
LIN {X 0,Y 256.124,Z 382.204,A -85,B 0,C 180,E1 -18664.033,E2 -18664.033} C_VEL
LIN {X 0,Y 256.113,Z 382.199,A -85,B 0,C 180,E1 -18667.269,E2 -18667.269} C_VEL
LIN {X 0,Y 256.063,Z 382.206,A -85,B 0,C 180,E1 -18672.178,E2 -18672.178} C_VEL
LIN {X 0,Y 256.027,Z 382.197,A -85,B 0,C 180,E1 -18676.664,E2 -18676.664} C_VEL
LIN {X 0,Y 256.045,Z 382.206,A -85,B 0,C 180,E1 -18680.852,E2 -18680.852} C_VEL
LIN {X 0,Y 256.081,Z 382.207,A -85,B 0,C 180,E1 -18684.806,E2 -18684.806} C_VEL
LIN {X 0,Y 256.086,Z 382.213,A -85,B 0,C 180,E1 -18688.57,E2 -18688.57} C_VEL
LIN {X 0,Y 256.084,Z 382.161,A -85,B 0,C 180,E1 -18692.188,E2 -18692.188} C_VEL
LIN {X 0,Y 256.087,Z 382.165,A -85,B 0,C 180,E1 -18695.69,E2 -18695.69} C_VEL
LIN {X 0,Y 256.147,Z 382.203,A -85,B 0,C 180,E1 -18699.102,E2 -18699.102} C_VEL
LIN {X 0,Y 256.16,Z 382.195,A -85,B 0,C 180,E1 -18700.809,E2 -18700.809} C_VEL
LIN {X 0,Y 255.457,Z 382.274,A -85,B 0,C 180,E1 -18702.122,E2 -18702.122} C_VEL
LIN {X 0,Y 252.617,Z 382.637,A -85,B 0,C 180,E1 -18704.265,E2 -18704.265} C_VEL
LIN {X 0,Y 250.248,Z 382.935,A -85,B 0,C 180,E1 -18706.009,E2 -18706.009} C_VEL
LIN {X 0,Y 249.258,Z 383.046,A -85,B 0,C 180,E1 -18707.36,E2 -18707.36} C_VEL
LIN {X 0,Y 249.19,Z 383.049,A -85,B 0,C 180,E1 -18707.817,E2 -18707.817} C_VEL
LIN {X 0,Y 249.437,Z 383.037,A -85,B 0,C 180,E1 -18711.901,E2 -18711.901} C_VEL
LIN {X 0,Y 249.264,Z 383.038,A -85,B 0,C 180,E1 -18715.147,E2 -18715.147} C_VEL
LIN {X 0,Y 249.663,Z 383.009,A -85,B 0,C 180,E1 -18718.386,E2 -18718.386} C_VEL
LIN {X 0,Y 249.664,Z 382.99,A -85,B 0,C 180,E1 -18721.612,E2 -18721.612} C_VEL
LIN {X 0,Y 249.429,Z 383.033,A -85,B 0,C 180,E1 -18726.471,E2 -18726.471} C_VEL
LIN {X 0,Y 249.343,Z 383.047,A -85,B 0,C 180,E1 -18729.736,E2 -18729.736} C_VEL
LIN {X 0,Y 249.159,Z 383.067,A -85,B 0,C 180,E1 -18734.705,E2 -18734.705} C_VEL
LIN {X 0,Y 249.114,Z 383.064,A -85,B 0,C 180,E1 -18738.079,E2 -18738.079} C_VEL
LIN {X 0,Y 249.085,Z 383.072,A -85,B 0,C 180,E1 -18741.518,E2 -18741.518} C_VEL
LIN {X 0,Y 249.086,Z 383.076,A -85,B 0,C 180,E1 -18745.459,E2 -18745.459} C_VEL
LIN {X 0,Y 249.037,Z 383.086,A -85,B 0,C 180,E1 -18748.973,E2 -18748.973} C_VEL
LIN {X 0,Y 249.027,Z 383.086,A -85,B 0,C 180,E1 -18752.426,E2 -18752.426} C_VEL
LIN {X 0,Y 249.01,Z 383.089,A -85,B 0,C 180,E1 -18756.348,E2 -18756.348} C_VEL
LIN {X 0,Y 248.971,Z 383.084,A -85,B 0,C 180,E1 -18760.484,E2 -18760.484} C_VEL
LIN {X 0,Y 248.997,Z 383.143,A -85,B 0,C 180,E1 -18762.435,E2 -18762.435} C_VEL
LIN {X 0,Y 250.798,Z 389.122,A -85,B 0,C 180,E1 -18764.812,E2 -18764.812} C_VEL
LIN {X 0,Y 257.137,Z 400.498,A -85,B 0,C 180,E1 -18766.426,E2 -18766.426} C_VEL
LIN {X 0,Y 264.751,Z 414.87,A -85,B 0,C 180,E1 -18768.246,E2 -18768.246} C_VEL
LIN {X 0,Y 272.226,Z 431.589,A -85,B 0,C 180,E1 -18769.982,E2 -18769.982} C_VEL
LIN {X 0,Y 277.73,Z 445.397,A -85,B 0,C 180,E1 -18771.225,E2 -18771.225} C_VEL
LIN {X 0,Y 278.635,Z 451.928,A -85,B 0,C 180,E1 -18771.555,E2 -18771.555} C_VEL
LIN {X 0,Y 274.148,Z 555.608,A -85,B 0,C 180,E1 -18774.153,E2 -18774.153} C_VEL
LIN {X 0,Y 272.756,Z 571.242,A -85,B 0,C 180,E1 -18774.793,E2 -18774.793} C_VEL
LIN {X 0,Y 270.677,Z 586.896,A -85,B 0,C 180,E1 -18775.729,E2 -18775.729} C_VEL
LIN {X 0,Y 268.231,Z 601.984,A -85,B 0,C 180,E1 -18776.975,E2 -18776.975} C_VEL
LIN {X 0,Y 265.502,Z 616.063,A -85,B 0,C 180,E1 -18778.48,E2 -18778.48} C_VEL
LIN {X 0,Y 262.411,Z 629.623,A -85,B 0,C 180,E1 -18780.299,E2 -18780.299} C_VEL
LIN {X 0,Y 259.679,Z 640.957,A -85,B 0,C 180,E1 -18782.169,E2 -18782.169} C_VEL
LIN {X 0,Y 256.928,Z 651.936,A -85,B 0,C 180,E1 -18784.375,E2 -18784.375} C_VEL
LIN {X 0,Y 254.412,Z 661.968,A -85,B 0,C 180,E1 -18786.818,E2 -18786.818} C_VEL
LIN {X 0,Y 251.895,Z 671.38,A -85,B 0,C 180,E1 -18789.589,E2 -18789.589} C_VEL
LIN {X 0,Y 250.028,Z 679.285,A -85,B 0,C 180,E1 -18792.446,E2 -18792.446} C_VEL
LIN {X 0,Y 248.608,Z 685.664,A -85,B 0,C 180,E1 -18795.26,E2 -18795.26} C_VEL
LIN {X 0,Y 247.531,Z 691.584,A -85,B 0,C 180,E1 -18798.536,E2 -18798.536} C_VEL
LIN {X 0,Y 247.084,Z 696.111,A -85,B 0,C 180,E1 -18801.824,E2 -18801.824} C_VEL
LIN {X 0,Y 246.92,Z 699.341,A -85,B 0,C 180,E1 -18805.102,E2 -18805.102} C_VEL
LIN {X 0,Y 246.963,Z 701.3,A -85,B 0,C 180,E1 -18808.369,E2 -18808.369} C_VEL
LIN {X 0,Y 246.952,Z 702.072,A -85,B 0,C 180,E1 -18811.631,E2 -18811.631} C_VEL
LIN {X 0,Y 246.843,Z 701.702,A -85,B 0,C 180,E1 -18814.9,E2 -18814.9} C_VEL
LIN {X 0,Y 247.033,Z 700.207,A -85,B 0,C 180,E1 -18818.178,E2 -18818.178} C_VEL
LIN {X 0,Y 247.664,Z 697.555,A -85,B 0,C 180,E1 -18821.457,E2 -18821.457} C_VEL
LIN {X 0,Y 248.923,Z 693.662,A -85,B 0,C 180,E1 -18824.72,E2 -18824.72} C_VEL
LIN {X 0,Y 250.763,Z 688.49,A -85,B 0,C 180,E1 -18827.956,E2 -18827.956} C_VEL
LIN {X 0,Y 253.397,Z 681.914,A -85,B 0,C 180,E1 -18831.134,E2 -18831.134} C_VEL
LIN {X 0,Y 256.259,Z 674.869,A -85,B 0,C 180,E1 -18833.861,E2 -18833.861} C_VEL
LIN {X 0,Y 259.276,Z 667.584,A -85,B 0,C 180,E1 -18836.198,E2 -18836.198} C_VEL
LIN {X 0,Y 263,Z 657.925,A -85,B 0,C 180,E1 -18838.751,E2 -18838.751} C_VEL
LIN {X 0,Y 267.478,Z 646.047,A -85,B 0,C 180,E1 -18841.261,E2 -18841.261} C_VEL
LIN {X 0,Y 271.818,Z 633.746,A -85,B 0,C 180,E1 -18843.328,E2 -18843.328} C_VEL
LIN {X 0,Y 275.557,Z 621.852,A -85,B 0,C 180,E1 -18844.955,E2 -18844.955} C_VEL
LIN {X 0,Y 278.805,Z 609.657,A -85,B 0,C 180,E1 -18846.325,E2 -18846.325} C_VEL
LIN {X 0,Y 281.758,Z 597.203,A -85,B 0,C 180,E1 -18847.445,E2 -18847.445} C_VEL
LIN {X 0,Y 284.693,Z 582.701,A -85,B 0,C 180,E1 -18848.447,E2 -18848.447} C_VEL
LIN {X 0,Y 286.997,Z 567.745,A -85,B 0,C 180,E1 -18849.205,E2 -18849.205} C_VEL
LIN {X 0,Y 288.575,Z 552.238,A -85,B 0,C 180,E1 -18849.739,E2 -18849.739} C_VEL
LIN {X 0,Y 293.584,Z 459.402,A -85,B 0,C 180,E1 -18851.963,E2 -18851.963} C_VEL
LIN {X 0,Y 287.641,Z 446.39,A -85,B 0,C 180,E1 -18853.667,E2 -18853.667} C_VEL
LIN {X 0,Y 281.505,Z 434.413,A -85,B 0,C 180,E1 -18855.512,E2 -18855.512} C_VEL
LIN {X 0,Y 273.907,Z 421.118,A -85,B 0,C 180,E1 -18857.963,E2 -18857.963} C_VEL
LIN {X 0,Y 266.879,Z 410.114,A -85,B 0,C 180,E1 -18860.442,E2 -18860.442} C_VEL
LIN {X 0,Y 262.967,Z 404.318,A -85,B 0,C 180,E1 -18861.935,E2 -18861.935} C_VEL
LIN {X 0,Y 259.14,Z 398.812,A -85,B 0,C 180,E1 -18863.491,E2 -18863.491} C_VEL
LIN {X 0,Y 254.916,Z 392.982,A -85,B 0,C 180,E1 -18865.345,E2 -18865.345} C_VEL
LIN {X 0,Y 250.869,Z 387.806,A -85,B 0,C 180,E1 -18867.264,E2 -18867.264} C_VEL
LIN {X 0,Y 250.381,Z 386.732,A -85,B 0,C 180,E1 -18867.631,E2 -18867.631} C_VEL
LIN {X 0,Y 249.023,Z 383.059,A -85,B 0,C 180,E1 -18870.33,E2 -18870.33} C_VEL
LIN {X 0,Y 249.103,Z 383.078,A -85,B 0,C 180,E1 -18874.964,E2 -18874.964} C_VEL
LIN {X 0,Y 249.094,Z 383.083,A -85,B 0,C 180,E1 -18878.603,E2 -18878.603} C_VEL
LIN {X 0,Y 249.243,Z 383.054,A -85,B 0,C 180,E1 -18883.623,E2 -18883.623} C_VEL
LIN {X 0,Y 249.236,Z 383.055,A -85,B 0,C 180,E1 -18888.616,E2 -18888.616} C_VEL
LIN {X 0,Y 249.419,Z 383.029,A -85,B 0,C 180,E1 -18891.901,E2 -18891.901} C_VEL
LIN {X 0,Y 249.278,Z 383.048,A -85,B 0,C 180,E1 -18895.149,E2 -18895.149} C_VEL
LIN {X 0,Y 249.67,Z 383.005,A -85,B 0,C 180,E1 -18898.388,E2 -18898.388} C_VEL
LIN {X 0,Y 249.664,Z 383.012,A -85,B 0,C 180,E1 -18901.614,E2 -18901.614} C_VEL
LIN {X 0,Y 249.421,Z 383.032,A -85,B 0,C 180,E1 -18906.61,E2 -18906.61} C_VEL
LIN {X 0,Y 249.345,Z 383.049,A -85,B 0,C 180,E1 -18909.737,E2 -18909.737} C_VEL
LIN {X 0,Y 249.208,Z 383.058,A -85,B 0,C 180,E1 -18914.704,E2 -18914.704} C_VEL
LIN {X 0,Y 249.138,Z 383.048,A -85,B 0,C 180,E1 -18918.078,E2 -18918.078} C_VEL
LIN {X 0,Y 249.027,Z 383.08,A -85,B 0,C 180,E1 -18922.123,E2 -18922.123} C_VEL
LIN {X 0,Y 249.689,Z 385.332,A -85,B 0,C 180,E1 -18922.552,E2 -18922.552} C_VEL
LIN {X 0,Y 251.514,Z 387.662,A -85,B 0,C 180,E1 -18923.466,E2 -18923.466} C_VEL
LIN {X 0,Y 253.515,Z 388.99,A -85,B 0,C 180,E1 -18924.355,E2 -18924.355} C_VEL
LIN {X 0,Y 255.419,Z 392.221,A -85,B 0,C 180,E1 -18925.273,E2 -18925.273} C_VEL
LIN {X 0,Y 257.912,Z 394.524,A -85,B 0,C 180,E1 -18926.319,E2 -18926.319} C_VEL
LIN {X 0,Y 260.274,Z 397.966,A -85,B 0,C 180,E1 -18927.326,E2 -18927.326} C_VEL
LIN {X 0,Y 262.001,Z 399.792,A -85,B 0,C 180,E1 -18927.998,E2 -18927.998} C_VEL
LIN {X 0,Y 264.981,Z 403.596,A -85,B 0,C 180,E1 -18929.141,E2 -18929.141} C_VEL
LIN {X 0,Y 272.466,Z 413.799,A -85,B 0,C 180,E1 -18931.801,E2 -18931.801} C_VEL
LIN {X 0,Y 278.548,Z 422.678,A -85,B 0,C 180,E1 -18933.771,E2 -18933.771} C_VEL
LIN {X 0,Y 283.628,Z 430.82,A -85,B 0,C 180,E1 -18935.318,E2 -18935.318} C_VEL
LIN {X 0,Y 291.154,Z 444.932,A -85,B 0,C 180,E1 -18937.499,E2 -18937.499} C_VEL
LIN {X 0,Y 294.021,Z 451.162,A -85,B 0,C 180,E1 -18938.308,E2 -18938.308} C_VEL
LIN {X 0,Y 288.89,Z 540.88,A -85,B 0,C 180,E1 -18940.414,E2 -18940.414} C_VEL
LIN {X 0,Y 287.396,Z 556.502,A -85,B 0,C 180,E1 -18941.017,E2 -18941.017} C_VEL
LIN {X 0,Y 285.363,Z 570.419,A -85,B 0,C 180,E1 -18941.782,E2 -18941.782} C_VEL
LIN {X 0,Y 282.696,Z 584.646,A -85,B 0,C 180,E1 -18942.829,E2 -18942.829} C_VEL
LIN {X 0,Y 279.703,Z 597.36,A -85,B 0,C 180,E1 -18944.007,E2 -18944.007} C_VEL
LIN {X 0,Y 276.403,Z 610.159,A -85,B 0,C 180,E1 -18945.524,E2 -18945.524} C_VEL
LIN {X 0,Y 272.74,Z 621.852,A -85,B 0,C 180,E1 -18947.185,E2 -18947.185} C_VEL
LIN {X 0,Y 268.842,Z 633.28,A -85,B 0,C 180,E1 -18949.191,E2 -18949.191} C_VEL
LIN {X 0,Y 264.902,Z 643.731,A -85,B 0,C 180,E1 -18951.43,E2 -18951.43} C_VEL
